	  ELSIF (#statStatus = #STATUS_COMMAND_ABORTED) AND (#statCommandAborted = FALSE) THEN // Commanded functionality has been aborted by another command
	    #statDone := FALSE;
	    #statBusy := FALSE;
	    #statActive := FALSE;
	    #statCommandAborted := TRUE;
	    #statError := FALSE;
	    #diagnostics.stateNumber := #statFBState;
	    #diagnostics.status := #statStatus;
	    #diagnostics.subFunctionStatus := #statSubfunctionStatus;
	    #diagnostics.additionalValue1 := #statAdditionalValue[1];
	    #diagnostics.additionalValue2 := #statAdditionalValue[2];
	    #statFBState := #FB_STATE_NO_PROCESSING; // Switch state machine to "no processing"
	    //Restore TO data
	    IF (#statReadyForNextCommand = FALSE) THEN
	      //only do if not done yet
	      "LKinCtrl_InitTODataRestore"(initTOData := #statInitTOData,
	                                   axesGroup := #axesGroup);
	    END_IF;
	    // Reset application specific outputs
	    #statReadyForNextCommand := FALSE;
	    #statCommandStep := #CMD_STEP_IDLE;
	    #statRemainingPathLength := -1.0;
	    
	  ELSIF (#tempExecute = FALSE) AND ((#statDone = TRUE) OR (#statError = TRUE) OR (#statCommandAborted = TRUE)) THEN // Reset outputs
	    #statDone := FALSE;
	    #statBusy := FALSE;
	    #statActive := FALSE;
	    #statCommandAborted := FALSE;
	    #statError := FALSE;
	    #statStatus := #STATUS_NO_CALL;
	    // Reset application specific outputs
	    #statReadyForNextCommand := FALSE;
	    #statCommandStep := #CMD_STEP_IDLE;
	    #statRemainingPathLength := -1.0;
	  END_IF;
	  
	  // Write static values to outputs
	  #done := #statDone;
	  #busy := #statBusy;
	  #active := #statActive;
	  #commandAborted := #statCommandAborted;
	  #error := #statError;
	  #status := #statStatus;
	  // Write application specific static values to outputs
	  #readyForNextCommand := #statReadyForNextCommand;
	  #commandStep := #statCommandStep;
	  #remainingPathLength := #statRemainingPathLength;
	END_REGION OUTPUTS
END_FUNCTION_BLOCK

FUNCTION "LKinCtrl_InitTODataStore" : "LKinCtrl_typePnPInitTOData"
TITLE = LKinCtrl_InitTODataStore
{ S7_Optimized_Access := 'TRUE' }
AUTHOR : 'handling.team.automation@siemens.com'
FAMILY : LKinCtrl
VERSION : 5.0
//Store specific TO data
   VAR_IN_OUT 
      axesGroup {InstructionName := 'TO_Kinematics'; LibVersion := '9.0'} : TO_Kinematics;   // Reference to axes group
   END_VAR


BEGIN
	//=============================================================================
	// SIEMENS AG
	// (c)Copyright 2023
	//-----------------------------------------------------------------------------
	// Library:       LKinCtrl
	// Tested with:   S7-1518TF-4 PN/DP, FW V3.1
	// Engineering:   TIA Portal V19
	// Restrictions:  ---
	// Requirements:  S7-1500T, FW V3.0
	// Functionality: Store specific TO data
	// Support: tech.team.motioncontrol@siemens.com
	// Note: Parameter comments are only available in language 'English (United States)'
	//-----------------------------------------------------------------------------
	// Change log table:
	// Version  Date       Expert in charge Changes applied
	// 01.00.00 21.09.2023 SF               First released version
	//=============================================================================
	
	//Blending length factor
	#LKinCtrl_InitTODataStore.factorBlendingLength := #axesGroup.Transition.FactorBlendingLength;
	//Orientation dynamics
	#LKinCtrl_InitTODataStore.orientationDefaults.velocity := #axesGroup.DynamicDefaults.Orientation.Velocity;
	#LKinCtrl_InitTODataStore.orientationDefaults.acceleration := #axesGroup.DynamicDefaults.Orientation.Acceleration;
	#LKinCtrl_InitTODataStore.orientationDefaults.deceleration := #axesGroup.DynamicDefaults.Orientation.Deceleration;
	#LKinCtrl_InitTODataStore.orientationDefaults.jerk := #axesGroup.DynamicDefaults.Orientation.Jerk;
END_FUNCTION

FUNCTION "LKinCtrl_CallMC_TrackConv" : Void
TITLE = LKinCtrl_CallMC_TrackConv
{ S7_Optimized_Access := 'TRUE' }
AUTHOR : 'handling.team.automation@siemens.com'
FAMILY : LKinCtrl
VERSION : 5.0
//Call given MC_TrackConveyorBelt instance
   VAR_INPUT 
      axis : DB_ANY;   // Axis input
      axesGroup {InstructionName := 'TO_Kinematics'; LibVersion := '9.0'} : TO_Kinematics;   // Kinematics input
   END_VAR

   VAR_IN_OUT 
      instTrackConveyorBelt {InstructionName := 'MC_TRACKCONVEYORBELT'; LibVersion := '9.0'} : MC_TRACKCONVEYORBELT;   // Instance of MC_TrackConveyorBelt to be called
   END_VAR

   VAR_TEMP 
      tempRefAxis {InstructionName := 'TO_PositioningAxis'; LibVersion := '9.0'} : REF_TO TO_PositioningAxis;   // Temporary reference to positioning axis
      tempRefEncoder {InstructionName := 'TO_ExternalEncoder'; LibVersion := '9.0'} : REF_TO TO_ExternalEncoder;   // Temporary reference to external encoder
      tempRefProxy {InstructionName := 'TO_LeadingAxisProxy'; LibVersion := '9.0'} : REF_TO TO_LeadingAxisProxy;   // Temporary reference to leading axis proxy
   END_VAR


BEGIN
	//================================================================================
	// SIEMENS AG
	// (c)Copyright 2023 All Rights Reserved
	//--------------------------------------------------------------------------------
	// Library: LKinCtrl
	// Tested with: S7-1517T-3 PN
	// Engineering: TIA Portal V18
	// Restrictions: -
	// Requirements: S7-1500T FW 3.0
	// Functionality: Call MC_TrackConveyorBelt
	// Support: tech.team.motioncontrol@siemens.com
	// Note: Parameter comments are only available in language 'English (United States)'
	//-----------------------------------------------------------------------------
	// Change log table:
	// Version    Date          Expert in charge    Changes applied
	// 01.00.00   11.01.2022    FR                  First released version
	//===========================================================================================
	
	CASE TypeOfDB(#axis) OF
	  TO_PositioningAxis, TO_SynchronousAxis:
	    #tempRefAxis ?= #axis;
	    IF #tempRefAxis = NULL THEN
	      // Error
	      RETURN;
	    END_IF;
	    
	    // call MC_TrackConveyorBelt
	    #instTrackConveyorBelt(AxesGroup := #axesGroup,
	                           ConveyorBelt := #tempRefAxis^);
	    
	  TO_ExternalEncoder:
	    #tempRefEncoder ?= #axis;
	    IF #tempRefEncoder = NULL THEN
	      // Error
	      RETURN;
	    END_IF;
	    
	    // call MC_TrackConveyorBelt
	    #instTrackConveyorBelt(AxesGroup := #axesGroup,
	                           ConveyorBelt := #tempRefEncoder^);
	    
	  TO_LeadingAxisProxy:
	    #tempRefProxy ?= #axis;
	    IF #tempRefProxy = NULL THEN
	      // Error
	      RETURN;
	    END_IF;
	    
	    // call MC_TrackConveyorBelt
	    #instTrackConveyorBelt(AxesGroup := #axesGroup,
	                           ConveyorBelt := #tempRefProxy^);
	    
	  ELSE
	    // invalid TO type
	    ;
	END_CASE;
	
	
END_FUNCTION

FUNCTION "LKinCtrl_CreateLinCmdSequence" : Word
TITLE = LKinCtrl_CreateLinCmdSequence
{ S7_Optimized_Access := 'TRUE' }
AUTHOR : 'handling.team.automation@siemens.com'
FAMILY : LKinCtrl
VERSION : 5.0
//Creation of the parameter for a linear command sequence
   VAR_INPUT 
      startParameter : "LKinCtrl_typePnPParameter";   // Depart vector parameter
      targetParameter : "LKinCtrl_typePnPParameter";   // Approach vector parameter
      position : Array[1..6] of LReal;   // Target position
      coordSystem : DInt;   // Target coordinate system, = 0: WCS, = 1: OCS[1], = 2: OCS[2], = 3: OCS[3]
      directionA : DInt;   // 1 - positive, 2 - negative, 3 - shortest way (Only necessary up to 4D Kinematics)
      bufferModeBegin : DInt;   // bufferMode for start of path motion
      transitionParameter : Array[1..5] of LReal;   // transitionParameter for start of path motion
      dynamics : "LKinCtrl_typePnPDynamics";   // Dynamics specification
      bufferModeTransition : DInt;   // bufferMode for blending post pick / pre target
      scaleMode : DInt;   // Scaling mode for start and target dynamics (0: disable, 1: velo, 2: velo and accel, 3: velo, accel and jerk)
   END_VAR

   VAR_OUTPUT 
      cmdPar : "LKinCtrl_typePnPLinCmdSeqParameter";   // Command parameters
      additionalValue : Array[1..5] of Word;   // Stati of subfunctions for diagnostics
   END_VAR

   VAR_IN_OUT 
      axesGroup {InstructionName := 'TO_Kinematics'; LibVersion := '9.0'} : TO_Kinematics;   // Reference to axes group
   END_VAR

   VAR_TEMP 
      tempUseStartDirection : Bool;
      tempUseTargetDirection : Bool;
      tempInt : Int;
      tempLreal : LReal;
      tempWord : Word;
      tempCase : Int;
      tempIntermStartPoint : Array[1..6] of LReal;
      tempIntermStartCoordSystem : DInt;
      tempIntermTargetPoint : Array[1..6] of LReal;
      tempIntermTargetCoordSystem : DInt;
      tempOrientationDimension : Int;
      tempStartPointFrame : "LKinCtrl_typeFrame";
      tempTargetPointFrame : "LKinCtrl_typeFrame";
      tempIntermPointFrame : "LKinCtrl_typeFrame";
      tempStartDirection : "LKinCtrl_typeCOff3DPoint";
      tempNormStartDirection : "LKinCtrl_typeCOff3DPoint";
      tempTargetDirection : "LKinCtrl_typeCOff3DPoint";
      tempNormTargetDirection : "LKinCtrl_typeCOff3DPoint";
      tempCmdPar : "LKinCtrl_typePnPLinCmdSeqParameter" := (((), [()], (), (), [-1.0], ((), (), ((), (), (), (), (), ()), ((), (), (), (), (), ())), (), ((), (), (), ()), (), ()), ((), [()], (), (), [-1.0], ((), (), ((), (), (), (), (), ()), ((), (), (), (), (), ())), (), ((), (), (), ()), (), ()), ((), [()], (), (), [-1.0], ((), (), ((), (), (), (), (), ()), ((), (), (), (), (), ())), (), ((), (), (), ()), (), ()), ((), [()], (), (), [-1.0], ((), (), ((), (), (), (), (), ()), ((), (), (), (), (), ())), (), ((), (), (), ()), (), ()), ((), [()], (), (), [-1.0], ((), (), ((), (), (), (), (), ()), ((), (), (), (), (), ())), (), ((), (), (), ()), (), ()), ());
      tempFactorBlendingLength : LReal;
      tempBlendingFromPreviousCmd : Bool;
      tempTransition1 : LReal;
      tempTransition2 : LReal;
      tempPossibleIntermTransition1 : LReal;
      tempPossibleIntermTransition2 : LReal;
      tempIntermTransition : LReal;
      tempAdditionalValue : Word;
      tempTimeOffset : LReal;
      tempEstimatedStartTransitionArea : LReal;
   END_VAR

   VAR CONSTANT 
      CASE_NO_VEC : Int := 1;   // Case: no start and target direction specified
      CASE_ONLY_TARGET_VEC : Int := 2;   // Case: only target direction specified
      CASE_ONLY_START_VEC : Int := 3;   // Case: only start direction specified
      CASE_ALL_VEC : Int := 4;   // Case: all directions specified
      INTERM_POINT_RATIO : LReal := 0.5;   // Intermediate point ratio
      STATUS_NO_ERR : Word := 16#0000;   // No error
      ERR_GET_TRACKING_INFO : Word := 16#9000;   // Error - Get tracking info
      ERR_BLENDING_NOT_ALLOWED : Word := 16#9001;   // Error - Blending is not allowed
      ERR_GET_ORI_DIMENSION : Word := 16#9002;   // Error - Get orientation dimension
      ERR_GET_LIN_POINT_DIST : Word := 16#9003;   // Error - Get linear point distance
      ERR_CALC_INTERM_POINT : Word := 16#9004;   // Error - Calculate intermediate point
      INTERM_POINT_MIN_BLENDING_FAC : LReal := 0.2;   // Minimum blending factor for intermediate point
      INTERM_POINT_MAX_BLENDING_FAC : LReal := 0.4;   // Maximum blending factor for intermediate point
   END_VAR


BEGIN
	//=============================================================================
	// SIEMENS AG
	// (c)Copyright 2023
	//-----------------------------------------------------------------------------
	// Library:       LKinCtrl
	// Tested with:   S7-1518TF-4 PN/DP, FW V3.1
	// Engineering:   TIA Portal V19
	// Restrictions:  ---
	// Requirements:  S7-1500T, FW V3.0
	// Functionality: This block is creating the parameter for a linear command sequence
	//                (Usage for LKinCtrl_MC_MovePickAndPlace...)
	// Support: tech.team.motioncontrol@siemens.com
	// Note: Parameter comments are only available in language 'English (United States)'
	//-----------------------------------------------------------------------------
	// Change log table:
	// Version  Date       Expert in charge Changes applied
	// 01.00.00 21.09.2023 SF               First released version
	//=============================================================================
	
	//Preset additional values
	FOR #tempInt := 1 TO 5 DO
	  #additionalValue[#tempInt] := #STATUS_NO_ERR;
	END_FOR;
	
	//Blending from previous command?
	#tempBlendingFromPreviousCmd := #bufferModeBegin <> "BM_BUFFERED";
	
	REGION GET_DIRECTION_INFO
	  //Save variable to vector data type
	  #tempStartDirection.x := #startParameter.direction[1];
	  #tempStartDirection.y := #startParameter.direction[2];
	  #tempStartDirection.z := #startParameter.direction[3];
	  //Get info about start vector
	  #tempUseStartDirection := NOT (#tempStartDirection.x = 0.0 AND #tempStartDirection.y = 0.0 AND #tempStartDirection.z = 0.0) AND #startParameter.workingHeight <> 0;
	  //Save variable to vector data type
	  #tempTargetDirection.x := #targetParameter.direction[1];
	  #tempTargetDirection.y := #targetParameter.direction[2];
	  #tempTargetDirection.z := #targetParameter.direction[3];
	  //Get info about target vector    
	  #tempUseTargetDirection := NOT (#tempTargetDirection.x = 0.0 AND #tempTargetDirection.y = 0.0 AND #tempTargetDirection.z = 0.0) AND #targetParameter.workingHeight <> 0;
	  
	  //Check if allowed
	  IF (#tempUseStartDirection = TRUE) AND (#tempBlendingFromPreviousCmd = TRUE) THEN
	    //not allowed
	    #LKinCtrl_CreateLinCmdSequence := #ERR_BLENDING_NOT_ALLOWED;
	    RETURN;
	  END_IF;
	  
	  //use target point in every case
	  #tempCmdPar.target.usePoint := TRUE;
	  
	  //Get info which points are used
	  IF (#tempUseStartDirection = FALSE) AND (#tempUseTargetDirection = FALSE) THEN
	    //No start and target direction specified
	    #tempCase := #CASE_NO_VEC;
	    //Set if points are used or not
	    #tempCmdPar.postStart.usePoint := FALSE;
	    #tempCmdPar.preTarget.usePoint := FALSE;
	    
	  ELSIF (#tempUseStartDirection = FALSE) THEN
	    //No start direction specified
	    #tempCase := #CASE_ONLY_TARGET_VEC;
	    //Set if points are used or not
	    #tempCmdPar.postStart.usePoint := FALSE;
	    #tempCmdPar.preTarget.usePoint := TRUE;
	    
	  ELSIF (#tempUseTargetDirection = FALSE) THEN
	    //No target direction specified
	    #tempCase := #CASE_ONLY_START_VEC;
	    //Set if points are used or not
	    #tempCmdPar.postStart.usePoint := TRUE;
	    #tempCmdPar.preTarget.usePoint := FALSE;
	    
	  ELSE
	    //All directions specified
	    #tempCase := #CASE_ALL_VEC;
	    //Set if points are used or not
	    #tempCmdPar.postStart.usePoint := TRUE;
	    #tempCmdPar.preTarget.usePoint := TRUE;
	    
	  END_IF;
	END_REGION REGION GET_DIRECTION_INFO
	
	REGION GET_START_INFO
	  //Get all start parameter depending on blending from previous cmd
	  //--> if blending would be active, kinematics would be still in motion
	  //--> start position and therefore the post start position cannot be determinded
	  IF (#tempBlendingFromPreviousCmd = FALSE) THEN
	    //Start point
	    //set parameter
	    #tempCmdPar.start.usePoint := TRUE; //Inidicates that parameter are valid
	    #tempCmdPar.start.directionA := #directionA;
	    #tempCmdPar.start.pathDynamics := #dynamics.path;
	    #tempCmdPar.start.dynamicAdaption := #dynamics.dynamicAdaption;
	    //get Start CS and tracking info 
	    #tempCmdPar.start.coordSystem := #axesGroup.StatusPath.CoordSystem;
	    #tempWord := "LKinCtrl_GetTrackingInfo"(coordSystem := #tempCmdPar.start.coordSystem,
	                                            axesGroup := #axesGroup,
	                                            trackingPar => #tempCmdPar.start.tracking);
	    IF (#tempWord.%X15 = TRUE) THEN
	      #LKinCtrl_CreateLinCmdSequence := #ERR_GET_TRACKING_INFO;
	      #additionalValue[1] := #tempWord;
	      RETURN;
	    END_IF;
	    //Start position
	    IF (#tempCmdPar.start.coordSystem = "CS_WCS") THEN
	      #tempCmdPar.start.position[1] := #axesGroup.TcpInWcs.x.Position;
	      #tempCmdPar.start.position[2] := #axesGroup.TcpInWcs.y.Position;
	      #tempCmdPar.start.position[3] := #axesGroup.TcpInWcs.z.Position;
	      #tempCmdPar.start.position[4] := #axesGroup.TcpInWcs.a.Position;
	      #tempCmdPar.start.position[5] := #axesGroup.TcpInWcs.b.Position;
	      #tempCmdPar.start.position[6] := #axesGroup.TcpInWcs.c.Position;
	    ELSIF (#tempCmdPar.start.coordSystem >= "CS_OCS1") AND (#tempCmdPar.start.coordSystem <= "CS_OCS3") THEN
	      #tempCmdPar.start.position[1] := #axesGroup.TcpInOcs[#tempCmdPar.start.coordSystem].x.Position;
	      #tempCmdPar.start.position[2] := #axesGroup.TcpInOcs[#tempCmdPar.start.coordSystem].y.Position;
	      #tempCmdPar.start.position[3] := #axesGroup.TcpInOcs[#tempCmdPar.start.coordSystem].z.Position;
	      #tempCmdPar.start.position[4] := #axesGroup.TcpInOcs[#tempCmdPar.start.coordSystem].a.Position;
	      #tempCmdPar.start.position[5] := #axesGroup.TcpInOcs[#tempCmdPar.start.coordSystem].b.Position;
	      #tempCmdPar.start.position[6] := #axesGroup.TcpInOcs[#tempCmdPar.start.coordSystem].c.Position;
	    END_IF;
	    
	    //PostStart point
	    IF (#tempCmdPar.postStart.usePoint = TRUE) THEN
	      //set parameter
	      #tempCmdPar.postStart.coordSystem := #tempCmdPar.start.coordSystem;
	      #tempCmdPar.postStart.directionA := #directionA;
	      #tempCmdPar.postStart.pathDynamics := "LKinCtrl_ScaleDynamics"(dynamicsIn := #dynamics.path,
	                                                                     scaleFactor := #startParameter.dynamicsFactor,
	                                                                     mode := #scaleMode);
	      #tempCmdPar.postStart.dynamicAdaption := #dynamics.dynamicAdaption;
	      #tempWord := "LKinCtrl_GetTrackingInfo"(coordSystem := #tempCmdPar.postStart.coordSystem,
	                                              axesGroup := #axesGroup,
	                                              trackingPar => #tempCmdPar.postStart.tracking);
	      IF (#tempWord.%X15 = TRUE) THEN
	        #LKinCtrl_CreateLinCmdSequence := #ERR_GET_TRACKING_INFO;
	        #additionalValue[1] := #tempWord;
	        RETURN;
	      END_IF;
	      //Norm start vector
	      IF (#tempUseStartDirection = TRUE) THEN
	        #tempNormStartDirection := "LKinCtrl_VecUnit"(#tempStartDirection);
	      ELSE
	        #tempNormStartDirection.x := 0.0;
	        #tempNormStartDirection.y := 0.0;
	        #tempNormStartDirection.z := 0.0;
	      END_IF;
	      //Calc point position
	      #tempCmdPar.postStart.position[1] := #tempCmdPar.start.position[1] + #tempNormStartDirection.x * (#startParameter.workingHeight); // + #start.transitionArea
	      #tempCmdPar.postStart.position[2] := #tempCmdPar.start.position[2] + #tempNormStartDirection.y * (#startParameter.workingHeight);
	      #tempCmdPar.postStart.position[3] := #tempCmdPar.start.position[3] + #tempNormStartDirection.z * (#startParameter.workingHeight);
	      #tempCmdPar.postStart.position[4] := #tempCmdPar.start.position[4];
	      #tempCmdPar.postStart.position[5] := #tempCmdPar.start.position[5];
	      #tempCmdPar.postStart.position[6] := #tempCmdPar.start.position[6];
	    END_IF;
	  ELSE
	    //Start parameter not valid
	    #tempCmdPar.start.usePoint := FALSE;
	  END_IF;
	END_REGION GET_START_INFO
	
	REGION GET_PRETARGET_INFO
	  //PreTarget point 
	  IF (#tempCmdPar.preTarget.usePoint = TRUE) THEN
	    //set parameter
	    //set buffer mode and transitionParameter below...
	    #tempCmdPar.preTarget.coordSystem := #coordSystem;
	    #tempCmdPar.preTarget.directionA := #directionA;
	    #tempCmdPar.preTarget.pathDynamics := #dynamics.path;
	    #tempCmdPar.preTarget.dynamicAdaption := #dynamics.dynamicAdaption;
	    #tempWord := "LKinCtrl_GetTrackingInfo"(coordSystem := #tempCmdPar.preTarget.coordSystem,
	                                            axesGroup := #axesGroup,
	                                            trackingPar => #tempCmdPar.preTarget.tracking);
	    IF (#tempWord.%X15 = TRUE) THEN
	      #LKinCtrl_CreateLinCmdSequence := #ERR_GET_TRACKING_INFO;
	      #additionalValue[1] := #tempWord;
	      RETURN;
	    END_IF;
	    //Norm start vector
	    IF (#tempUseTargetDirection = TRUE) THEN
	      #tempNormTargetDirection := "LKinCtrl_VecUnit"(#tempTargetDirection);
	    ELSE
	      #tempNormTargetDirection.x := 0.0;
	      #tempNormTargetDirection.y := 0.0;
	      #tempNormTargetDirection.z := 0.0;
	    END_IF;
	    //Calc point position
	    #tempCmdPar.preTarget.position[1] := #position[1] + #tempNormTargetDirection.x * (#targetParameter.workingHeight);
	    #tempCmdPar.preTarget.position[2] := #position[2] + #tempNormTargetDirection.y * (#targetParameter.workingHeight);
	    #tempCmdPar.preTarget.position[3] := #position[3] + #tempNormTargetDirection.z * (#targetParameter.workingHeight);
	    #tempCmdPar.preTarget.position[4] := #position[4];
	    #tempCmdPar.preTarget.position[5] := #position[5];
	    #tempCmdPar.preTarget.position[6] := #position[6];
	  END_IF;
	END_REGION GET_PRETARGET_INFO
	
	REGION GET_TARGET_INFO
	  //Target point
	  IF (#tempCmdPar.target.usePoint = TRUE) THEN
	    //set parameter
	    //set path dynamics, buffer mode and transitionParameter below...
	    #tempCmdPar.target.coordSystem := #coordSystem;
	    #tempCmdPar.target.directionA := #directionA;
	    #tempCmdPar.target.dynamicAdaption := #dynamics.dynamicAdaption;
	    #tempWord := "LKinCtrl_GetTrackingInfo"(coordSystem := #tempCmdPar.target.coordSystem,
	                                            axesGroup := #axesGroup,
	                                            trackingPar => #tempCmdPar.target.tracking);
	    IF (#tempWord.%X15 = TRUE) THEN
	      #LKinCtrl_CreateLinCmdSequence := #ERR_GET_TRACKING_INFO;
	      #additionalValue[1] := #tempWord;
	      RETURN;
	    END_IF;
	    #tempCmdPar.target.position := #position;
	  END_IF;
	END_REGION GET_TARGET_INFO
	
	REGION GET_INTERMEDIATE_INFO
	  //Check if intermediate point is necessary (motion between two tracked OCS)??
	  IF (#tempCmdPar.start.tracking.active = TRUE)
	    AND (#tempCmdPar.target.tracking.active = TRUE)
	    AND (#tempCmdPar.start.coordSystem <> #tempCmdPar.target.coordSystem)
	    AND (#tempCmdPar.start.coordSystem >= "CS_OCS1") AND (#tempCmdPar.start.coordSystem <= "CS_OCS3")
	    AND (#tempCmdPar.target.coordSystem >= "CS_OCS1") AND (#tempCmdPar.target.coordSystem <= "CS_OCS3")
	  THEN
	    IF (#tempBlendingFromPreviousCmd = TRUE) THEN
	      //not allowed
	      #LKinCtrl_CreateLinCmdSequence := #ERR_BLENDING_NOT_ALLOWED;
	      RETURN;
	    END_IF;
	    
	    //set parameter
	    //set buffer mode and transitionParameter below...
	    #tempCmdPar.intermediate.usePoint := TRUE;
	    #tempCmdPar.intermediate.coordSystem := "CS_WCS";
	    #tempCmdPar.intermediate.directionA := #tempCmdPar.target.directionA;
	    #tempCmdPar.intermediate.pathDynamics := #dynamics.path;
	    #tempCmdPar.intermediate.dynamicAdaption := #dynamics.dynamicAdaption;
	    
	    //set values for point calculation
	    IF (#tempCmdPar.postStart.usePoint = TRUE) THEN
	      #tempIntermStartPoint := #tempCmdPar.postStart.position;
	      #tempIntermStartCoordSystem := #tempCmdPar.postStart.coordSystem;
	    ELSE
	      #tempIntermStartPoint := #tempCmdPar.start.position;
	      #tempIntermStartCoordSystem := #tempCmdPar.start.coordSystem;
	    END_IF;
	    
	    IF (#tempCmdPar.preTarget.usePoint = TRUE) THEN
	      #tempIntermTargetPoint := #tempCmdPar.preTarget.position;
	      #tempIntermTargetCoordSystem := #tempCmdPar.preTarget.coordSystem;
	    ELSE
	      #tempIntermTargetPoint := #tempCmdPar.target.position;
	      #tempIntermTargetCoordSystem := #tempCmdPar.target.coordSystem;
	    END_IF;
	    
	    //get ori dimension according to kinematics
	    #tempWord := "LKinCtrl_GetOrientationDimension"(orientationDimension => #tempOrientationDimension,
	                                                    axesGroup := #axesGroup);
	    IF (#tempWord.%X15 = TRUE) THEN
	      #LKinCtrl_CreateLinCmdSequence := #ERR_GET_ORI_DIMENSION;
	      #additionalValue[1] := #tempWord;
	      RETURN;
	    END_IF;
	    
	    //Set additional time duration for reaching start point (= post start)
	    IF (#tempCmdPar.postStart.usePoint = TRUE) THEN
	      // Estimated transition area around post start
	      #tempEstimatedStartTransitionArea := LIMIT(MN := 0.0, IN := #startParameter.transitionArea, MX := #startParameter.workingHeight);
	      // Calc time for motion between start and post start
	      #tempWord := "LKinCtrl_PositioningTime"(distance := #startParameter.workingHeight, //Use complete length 
	                                              velocity := #tempCmdPar.postStart.pathDynamics.velocity * #axesGroup.Override.Velocity / 100.0,
	                                              acceleration := #tempCmdPar.postStart.pathDynamics.acceleration,
	                                              deceleration := #tempCmdPar.postStart.pathDynamics.deceleration,
	                                              jerk := #tempCmdPar.postStart.pathDynamics.jerk,
	                                              "time" => #tempTimeOffset);
	      //Fracture time - better estimation than calculate time with standstill at start of blending 
	      #tempTimeOffset := #tempTimeOffset * (1.0 - #tempEstimatedStartTransitionArea / #startParameter.workingHeight);
	      //Reset time if error occured
	      IF (#tempWord.%X15 = TRUE) THEN
	        #tempTimeOffset := 0.0;
	      END_IF;
	    ELSE
	      //No additional time
	      #tempTimeOffset := 0.0;
	      #tempEstimatedStartTransitionArea := 0.0;
	    END_IF;
	    
	    //calculate point
	    #tempWord := "LKinCtrl_CalcIntermediatePoint"(startPosition := #tempIntermStartPoint,
	                                                  targetPosition := #tempIntermTargetPoint,
	                                                  startCoordSystem := #tempIntermStartCoordSystem,
	                                                  targetCoordSystem := #tempIntermTargetCoordSystem,
	                                                  ratio := #INTERM_POINT_RATIO,
	                                                  orientationDimension := #tempOrientationDimension,
	                                                  directionA := #tempCmdPar.intermediate.directionA,
	                                                  pathDynamics := #tempCmdPar.intermediate.pathDynamics,
	                                                  timeOffset := #tempTimeOffset,
	                                                  intermediatePosition => #tempCmdPar.intermediate.position,
	                                                  additionalValue => #tempAdditionalValue,
	                                                  axesGroup := #axesGroup);
	    IF (#tempWord.%X15 = TRUE) THEN
	      #LKinCtrl_CreateLinCmdSequence := #ERR_CALC_INTERM_POINT;
	      #additionalValue[1] := #tempWord;
	      #additionalValue[2] := #tempAdditionalValue;
	      RETURN;
	    END_IF;
	  ELSE
	    #tempCmdPar.intermediate.usePoint := FALSE;
	  END_IF;
	END_REGION GET_INTERMEDIATE_INFO
	
	REGION CALC_LIN_POINT_DISTANCE
	  //Calc distance to previous point
	  #tempWord := "LKinCtrl_GetDistanceToPrevious"(cmdPar := #tempCmdPar,
	                                                axesGroup := #axesGroup);
	  IF (#tempWord.%X15 = TRUE) THEN
	    #LKinCtrl_CreateLinCmdSequence := #ERR_GET_LIN_POINT_DIST;
	    #additionalValue[1] := #tempWord;
	    RETURN;
	  END_IF;
	END_REGION CALC_LIN_POINT_DISTANCE
	
	REGION CALC_BLENDING_INFO
	  //get blending info and calc radii for all point
	  CASE #tempCase OF
	      
	    #CASE_NO_VEC:
	      
	      REGION BLENDING_NO_VEC
	        //Set path dynamics for target
	        #tempCmdPar.target.pathDynamics := #dynamics.path;
	        //Intermediate point necessary?
	        IF (#tempCmdPar.intermediate.usePoint = TRUE) THEN
	          //info: 3
	          //No blending from previous motion!
	          //Start to intermediate
	          #tempCmdPar.intermediate.bufferMode := "BM_BUFFERED";
	          //Blend to target with max radius (100%!)
	          #tempCmdPar.target.bufferMode := #bufferModeTransition;
	          #tempCmdPar.target.transitionParameter[1] := #tempCmdPar.target.distanceToPrevious * #INTERM_POINT_MAX_BLENDING_FAC;
	        ELSE
	          //info: 1 & 9
	          //Blend to target with start specification
	          #tempCmdPar.target.bufferMode := #bufferModeBegin;
	          #tempCmdPar.target.transitionParameter := #transitionParameter;
	        END_IF;
	      END_REGION BLENDING_NO_VEC
	      
	    #CASE_ONLY_TARGET_VEC:
	      
	      REGION BLENDING_ONLY_TARGET_VEC
	        //Set path dynamics for target
	        #tempCmdPar.target.pathDynamics := "LKinCtrl_ScaleDynamics"(dynamicsIn := #dynamics.path,
	                                                                    scaleFactor := #targetParameter.dynamicsFactor,
	                                                                    mode := #scaleMode);
	        
	        //Intermediate point necessary?
	        IF (#tempCmdPar.intermediate.usePoint = TRUE) THEN
	          //info: 4
	          //No blending from previous motion!
	          //Start to intermediate
	          #tempCmdPar.intermediate.bufferMode := "BM_BUFFERED";
	          //Blend to pretarget with max radius
	          //Get radius
	          #tempCmdPar.preTarget.bufferMode := #bufferModeTransition;
	          //is target transition overlaping minimum intermediate radius?
	          IF (#targetParameter.transitionArea > (1.0 - #INTERM_POINT_MIN_BLENDING_FAC) * #tempCmdPar.preTarget.distanceToPrevious) THEN
	            //yes - shorten transition area
	            #tempTransition1 := (1.0 - #INTERM_POINT_MIN_BLENDING_FAC) * #tempCmdPar.preTarget.distanceToPrevious;
	          ELSE
	            //no - use transition area from spec
	            #tempTransition1 := #targetParameter.transitionArea;
	          END_IF;
	          #tempCmdPar.preTarget.transitionParameter[1] := MIN(IN1 := #tempCmdPar.preTarget.distanceToPrevious - #tempTransition1, IN2 := #tempCmdPar.preTarget.distanceToPrevious * #INTERM_POINT_MAX_BLENDING_FAC);
	          //Blend to target with specified transition area
	          IF (#targetParameter.transitionArea <> 0.0) THEN
	            #tempCmdPar.target.bufferMode := #bufferModeTransition;
	            #tempCmdPar.target.transitionParameter[1] := #tempTransition1; //use from calculation above
	          ELSE
	            #tempCmdPar.target.bufferMode := "BM_BUFFERED";
	          END_IF;
	        ELSE
	          //info: 2 & 10
	          //Blend to pretarget with start specification
	          #tempCmdPar.preTarget.bufferMode := #bufferModeBegin;
	          #tempCmdPar.preTarget.transitionParameter[1] := #transitionParameter[1];
	          //Blend to target with specified transition area
	          IF (#targetParameter.transitionArea <> 0.0) THEN
	            #tempCmdPar.target.bufferMode := #bufferModeTransition;
	            #tempCmdPar.target.transitionParameter[1] := #targetParameter.transitionArea;
	          ELSE
	            #tempCmdPar.target.bufferMode := "BM_BUFFERED";
	          END_IF;
	        END_IF;
	      END_REGION BLENDING_ONLY_TARGET_VEC
	      
	    #CASE_ONLY_START_VEC:
	      //Always start from standstill, no blending from previous motion
	      
	      REGION BLENDING_ONLY_START_VEC
	        //Set path dynamics for target
	        #tempCmdPar.target.pathDynamics := #dynamics.path;
	        
	        //Intermediate point necessary?
	        IF (#tempCmdPar.intermediate.usePoint = TRUE) THEN
	          //info: 7
	          //no blending to post start
	          #tempCmdPar.postStart.bufferMode := "BM_BUFFERED";
	          //is start transition overlaping minimum intermediate radius?
	          IF (#startParameter.transitionArea > (1.0 - #INTERM_POINT_MIN_BLENDING_FAC) * #tempCmdPar.target.distanceToPrevious) THEN
	            //yes - shorten transition area
	            #tempTransition1 := (1.0 - #INTERM_POINT_MIN_BLENDING_FAC) * #tempCmdPar.target.distanceToPrevious;
	          ELSE
	            //no - use transition area from spec
	            #tempTransition1 := #startParameter.transitionArea;
	          END_IF;
	          IF (#startParameter.transitionArea <> 0.0) THEN
	            #tempCmdPar.intermediate.bufferMode := #bufferModeTransition;
	            #tempCmdPar.intermediate.transitionParameter[1] := #tempTransition1;
	          ELSE
	            #tempCmdPar.intermediate.bufferMode := "BM_BUFFERED";
	          END_IF;
	          //Blend to target with resulting radius
	          #tempCmdPar.target.bufferMode := #bufferModeTransition;
	          #tempCmdPar.target.transitionParameter[1] := MIN(IN1 := #tempCmdPar.target.distanceToPrevious - #tempTransition1, IN2 := #tempCmdPar.target.distanceToPrevious * #INTERM_POINT_MAX_BLENDING_FAC);
	        ELSE
	          //info: 5
	          //no blending to post start
	          #tempCmdPar.postStart.bufferMode := "BM_BUFFERED";
	          //Blend to target with start transition area
	          IF (#startParameter.transitionArea <> 0.0) THEN
	            #tempCmdPar.target.bufferMode := #bufferModeTransition;
	            #tempCmdPar.target.transitionParameter[1] := #startParameter.transitionArea;
	          ELSE
	            #tempCmdPar.target.bufferMode := "BM_BUFFERED";
	          END_IF;
	        END_IF;
	      END_REGION REGION BLENDING_ONLY_START_VEC
	      
	    #CASE_ALL_VEC:
	      //Always Start from standstill, no blending from previous motion
	      
	      REGION BLENDING_ALL_VEC
	        //Set path dynamics for target
	        #tempCmdPar.target.pathDynamics := "LKinCtrl_ScaleDynamics"(dynamicsIn := #dynamics.path,
	                                                                    scaleFactor := #targetParameter.dynamicsFactor,
	                                                                    mode := #scaleMode);
	        
	        //Intermediate point necessary?
	        IF (#tempCmdPar.intermediate.usePoint = TRUE) THEN
	          //info: 8
	          //no blending to post start
	          #tempCmdPar.postStart.bufferMode := "BM_BUFFERED";
	          
	          //is start transition overlaping minimum intermediate radius?
	          IF (#startParameter.transitionArea > (1.0 - #INTERM_POINT_MIN_BLENDING_FAC) * #tempCmdPar.intermediate.distanceToPrevious) THEN
	            //yes - shorten transition area
	            #tempTransition1 := (1.0 - #INTERM_POINT_MIN_BLENDING_FAC) * #tempCmdPar.intermediate.distanceToPrevious;
	          ELSE
	            //no - use transition area from spec
	            #tempTransition1 := #startParameter.transitionArea;
	          END_IF;
	          #tempPossibleIntermTransition1 := MIN(IN1 := #tempCmdPar.intermediate.distanceToPrevious - #tempTransition1, IN2 := #tempCmdPar.intermediate.distanceToPrevious * #INTERM_POINT_MAX_BLENDING_FAC);
	          
	          //is target transition overlaping minimum intermediate radius?
	          IF (#targetParameter.transitionArea > (1.0 - #INTERM_POINT_MIN_BLENDING_FAC) * #tempCmdPar.preTarget.distanceToPrevious) THEN
	            //yes - shorten transition area
	            #tempTransition2 := (1.0 - #INTERM_POINT_MIN_BLENDING_FAC) * #tempCmdPar.preTarget.distanceToPrevious;
	          ELSE
	            //no - use transition area from spec
	            #tempTransition2 := #targetParameter.transitionArea;
	          END_IF;
	          #tempPossibleIntermTransition2 := MIN(IN1 := #tempCmdPar.preTarget.distanceToPrevious - #tempTransition2, IN2 := #tempCmdPar.preTarget.distanceToPrevious * #INTERM_POINT_MAX_BLENDING_FAC);
	          
	          //Get minimum intermediate transition
	          #tempIntermTransition := MIN(IN1 := #tempPossibleIntermTransition1, IN2 := #tempPossibleIntermTransition2);
	          //adapt 1st if necessary
	          #tempTransition1 := MIN(IN1 := #tempTransition1, IN2 := #tempCmdPar.intermediate.distanceToPrevious - #tempIntermTransition);
	          //adapt 2nd if necessary
	          #tempTransition2 := MIN(IN1 := #tempTransition2, IN2 := #tempCmdPar.preTarget.distanceToPrevious - #tempIntermTransition);
	          
	          //Blend to intermediate with start transition area
	          IF (#startParameter.transitionArea <> 0.0) THEN
	            #tempCmdPar.intermediate.bufferMode := #bufferModeTransition;
	            #tempCmdPar.intermediate.transitionParameter[1] := #tempTransition1;
	          ELSE
	            #tempCmdPar.intermediate.bufferMode := "BM_BUFFERED";
	          END_IF;
	          
	          //Blend to pretarget with intermediate radius
	          #tempCmdPar.preTarget.bufferMode := #bufferModeTransition;
	          #tempCmdPar.preTarget.transitionParameter[1] := #tempIntermTransition;
	          //Blend to target with target transition area
	          IF (#targetParameter.transitionArea <> 0.0) THEN
	            #tempCmdPar.target.bufferMode := #bufferModeTransition;
	            #tempCmdPar.target.transitionParameter[1] := #tempTransition2;
	          ELSE
	            #tempCmdPar.target.bufferMode := "BM_BUFFERED";
	          END_IF;
	        ELSE
	          //info: 6
	          //no blending to post start
	          #tempCmdPar.postStart.bufferMode := "BM_BUFFERED";
	          //Check if blending radii are overlapping
	          IF ((#startParameter.transitionArea + #targetParameter.transitionArea) > #tempCmdPar.preTarget.distanceToPrevious)
	            AND ((#startParameter.transitionArea + #targetParameter.transitionArea) <> 0.0)
	          THEN
	            //Yes - shorten both radi by overplapping factor
	            #tempTransition1 := #startParameter.transitionArea * #tempCmdPar.preTarget.distanceToPrevious / (#startParameter.transitionArea + #targetParameter.transitionArea);
	            #tempTransition2 := #targetParameter.transitionArea * #tempCmdPar.preTarget.distanceToPrevious / (#startParameter.transitionArea + #targetParameter.transitionArea);
	          ELSE
	            //No - set areas directly
	            #tempTransition1 := #startParameter.transitionArea;
	            #tempTransition2 := #targetParameter.transitionArea;
	          END_IF;
	          //Blend to pretarget with start transition area
	          IF (#startParameter.transitionArea <> 0.0) THEN
	            #tempCmdPar.preTarget.bufferMode := #bufferModeTransition;
	            #tempCmdPar.preTarget.transitionParameter[1] := #tempTransition1;
	          ELSE
	            #tempCmdPar.preTarget.bufferMode := "BM_BUFFERED";
	          END_IF;
	          //Blend to target with target transition area
	          IF (#targetParameter.transitionArea <> 0.0) THEN
	            #tempCmdPar.target.bufferMode := #bufferModeTransition;
	            #tempCmdPar.target.transitionParameter[1] := #tempTransition2;
	          ELSE
	            #tempCmdPar.target.bufferMode := "BM_BUFFERED";
	          END_IF;
	        END_IF;
	      END_REGION BLENDING_ALL_VEC
	      
	    ELSE
	      ;
	  END_CASE;
	  
	END_REGION CALC_BLENDING_INFO
	
	REGION GET_NUMBER_OF_USED_CMD
	  //init value
	  #tempCmdPar.numberOfUsedCmd := 0;
	  IF (#tempCmdPar.postStart.usePoint = TRUE) THEN
	    #tempCmdPar.numberOfUsedCmd += 1;
	  END_IF;
	  IF (#tempCmdPar.intermediate.usePoint = TRUE) THEN
	    #tempCmdPar.numberOfUsedCmd += 1;
	  END_IF;
	  IF (#tempCmdPar.preTarget.usePoint = TRUE) THEN
	    #tempCmdPar.numberOfUsedCmd += 1;
	  END_IF;
	  IF (#tempCmdPar.target.usePoint = TRUE) THEN
	    #tempCmdPar.numberOfUsedCmd += 1;
	  END_IF;
	END_REGION GET_NUMBER_OF_USED_CMD
	
	REGION OUTPUT
	  //Everything done - copy to Out var
	  #cmdPar := #tempCmdPar;
	  #LKinCtrl_CreateLinCmdSequence := #STATUS_NO_ERR;
	END_REGION OUTPUT
	
	
END_FUNCTION

FUNCTION "LKinCtrl_GetTrackingInfo" : Word
TITLE = LKinCtrl_GetTrackingInfo
{ S7_Optimized_Access := 'TRUE' }
AUTHOR : 'handling.team.automation@siemens.com'
FAMILY : LKinCtrl
VERSION : 5.0
//Get information about active conveyor tracking on specific OCS
   VAR_INPUT 
      coordSystem : DInt;   // Coordiante system to be checked
   END_VAR

   VAR_OUTPUT 
      trackingPar : "LKinCtrl_typePnPTrackingProperties";   // Tracking info
   END_VAR

   VAR_IN_OUT 
      axesGroup {InstructionName := 'TO_Kinematics'; LibVersion := '9.0'} : TO_Kinematics;   // Reference to axes group
   END_VAR

   VAR_TEMP 
      tempInt : Int;
      tempLreal : LReal;
      tempWord : Word;
   END_VAR

   VAR CONSTANT 
      STATUS_NO_ERR : Word := 16#0000;   // No error
      ERR_GET_AXIS_MOTION_VEC : Word := 16#8000;   // Error - Get axis motion vector
   END_VAR


BEGIN
	//=============================================================================
	// SIEMENS AG
	// (c)Copyright 2023
	//-----------------------------------------------------------------------------
	// Library:       LKinCtrl
	// Tested with:   S7-1518TF-4 PN/DP, FW V3.1
	// Engineering:   TIA Portal V19
	// Restrictions:  ---
	// Requirements:  S7-1500T, FW V3.0
	// Functionality: This block returns information about active conveyor tracking of a OCS
	//                (Usage for LKinCtrl_MC_MovePickAndPlace...)
	// Support: tech.team.motioncontrol@siemens.com
	// Note: Parameter comments are only available in language 'English (United States)'
	//-----------------------------------------------------------------------------
	// Change log table:
	// Version  Date       Expert in charge Changes applied
	// 01.00.00 21.09.2023 SF               First released version
	//=============================================================================
	
	#LKinCtrl_GetTrackingInfo := #STATUS_NO_ERR;
	//preset active as false
	#trackingPar.active := FALSE;
	
	FOR #tempInt := "CS_OCS1" TO "CS_OCS3" DO
	  IF (#coordSystem = #tempInt) THEN
	    IF (#axesGroup.StatusConveyor[#tempInt].TrackingState > 0) THEN
	      //Tracking on start is actvie
	      #trackingPar.active := TRUE;
	      //Get CS frame (one by one due to system...)
	      #trackingPar.frame.x := #axesGroup.StatusOcsFrame[#tempInt].x;
	      #trackingPar.frame.y := #axesGroup.StatusOcsFrame[#tempInt].y;
	      #trackingPar.frame.z := #axesGroup.StatusOcsFrame[#tempInt].z;
	      #trackingPar.frame.a := #axesGroup.StatusOcsFrame[#tempInt].a;
	      #trackingPar.frame.b := #axesGroup.StatusOcsFrame[#tempInt].b;
	      #trackingPar.frame.c := #axesGroup.StatusOcsFrame[#tempInt].c;
	      //Get Obj position (one by one due to system...)
	      #trackingPar.objectPosition.x := #axesGroup.StatusConveyor[#tempInt].ObjectPosition.x;
	      #trackingPar.objectPosition.y := #axesGroup.StatusConveyor[#tempInt].ObjectPosition.y;
	      #trackingPar.objectPosition.z := #axesGroup.StatusConveyor[#tempInt].ObjectPosition.z;
	      #trackingPar.objectPosition.a := #axesGroup.StatusConveyor[#tempInt].ObjectPosition.a;
	      #trackingPar.objectPosition.b := #axesGroup.StatusConveyor[#tempInt].ObjectPosition.b;
	      #trackingPar.objectPosition.c := #axesGroup.StatusConveyor[#tempInt].ObjectPosition.c;
	      //Get conveyor axis motion values
	      #tempWord := "LKinCtrl_GetAxisMotionVec"(actualValues := FALSE,
	                                               position => #tempLreal,
	                                               velocity => #trackingPar.velocity,
	                                               acceleration => #tempLreal,
	                                               axis := #axesGroup.StatusConveyor[#tempInt].ConveyorBelt);
	      IF (#tempWord.%X15 = TRUE) THEN
	        #LKinCtrl_GetTrackingInfo := #ERR_GET_AXIS_MOTION_VEC;
	        RETURN; //TODO use EXIT for performance?
	      END_IF;
	      RETURN; //TODO use EXIT for performance?
	    ELSE
	      #trackingPar.active := FALSE;
	    END_IF;
	  END_IF;
	END_FOR;
END_FUNCTION

FUNCTION "LKinCtrl_GetAxisMotionVec" : Word
TITLE = LKinCtrl_GetAxisMotionVec
{ S7_Optimized_Access := 'TRUE' }
AUTHOR : 'handling.team.automation@siemens.com'
FAMILY : LKinCtrl
VERSION : 5.0
//Get axes motion vector (position, velocity, acceleration) of positioning axis / synchronous axis
   VAR_INPUT 
      actualValues : Bool;   // TRUE: Get actual axis values
      axis : DB_ANY;   // Reference to axis DB
   END_VAR

   VAR_OUTPUT 
      position : LReal;   // Axis position
      velocity : LReal;   // Axis velocity
      acceleration : LReal;   // Axis acceleration
   END_VAR

   VAR_TEMP 
      tempRefToPosAxis {InstructionName := 'TO_PositioningAxis'; LibVersion := '9.0'} : REF_TO TO_PositioningAxis;
   END_VAR

   VAR CONSTANT 
      STATUS_NO_ERR : Word := 16#0000;   // No error
      ERR_AXIS_TYPE : Word := 16#8000;   // Error - Invalid axis type (< PosAxis)
   END_VAR


BEGIN
	//=============================================================================
	// SIEMENS AG
	// (c)Copyright 2023
	//-----------------------------------------------------------------------------
	// Library:       LKinCtrl
	// Tested with:   S7-1518TF-4 PN/DP, FW V3.1
	// Engineering:   TIA Portal V19
	// Restrictions:  ---
	// Requirements:  S7-1500T, FW V3.0
	// Functionality: This block is returning the motion vector (position, velocity, acceleration)
	//                of an positioning axis / synchronous axis
	// Support: tech.team.motioncontrol@siemens.com
	// Note: Parameter comments are only available in language 'English (United States)'
	//-----------------------------------------------------------------------------
	// Change log table:
	// Version  Date       Expert in charge Changes applied
	// 01.00.00 21.09.2023 SF               First released version
	//=============================================================================
	
	//Preset output
	#LKinCtrl_GetAxisMotionVec := #STATUS_NO_ERR;
	
	//Axis type at least pos axis?
	#tempRefToPosAxis ?= #axis;
	
	IF (#tempRefToPosAxis <> NULL) THEN
	  //get actual or setpoint values?
	  IF (#actualValues = TRUE) THEN
	    #position := #tempRefToPosAxis^.ActualPosition;
	    #velocity := #tempRefToPosAxis^.ActualVelocity;
	    #acceleration := #tempRefToPosAxis^.ActualAcceleration;
	  ELSE
	    #position := #tempRefToPosAxis^.Position;
	    #velocity := #tempRefToPosAxis^.Velocity;
	    #acceleration := #tempRefToPosAxis^.Acceleration;
	  END_IF;
	ELSE
	  #LKinCtrl_GetAxisMotionVec := #ERR_AXIS_TYPE;
	END_IF;
	
	
END_FUNCTION

FUNCTION "LKinCtrl_ScaleDynamics" : "LKinCtrl_typePathDynamics"
TITLE = LKinCtrl_ScaleDynamics
{ S7_Optimized_Access := 'TRUE' }
AUTHOR : 'handling.team.automation@siemens.com'
FAMILY : LKinCtrl
VERSION : 5.0
//Scale dynamics values according to input factor
   VAR_INPUT 
      dynamicsIn : "LKinCtrl_typePathDynamics";   // Input dynamics
      scaleFactor : LReal;   // Scaling factor
      mode : DInt;   // Scaling mode for start and target dynamics (0: disable, 1: velo, 2: velo and accel, 3: velo, accel and jerk)
   END_VAR

   VAR CONSTANT 
      MODE_VELO_ACCEL : DInt := 2;   // Scale only velocity and acceleration
      MODE_VELO : DInt := 1;   // Scale only velocity
      MODE_DISALBE : DInt := 0;   // Scale nothing
   END_VAR


BEGIN
	//=============================================================================
	// SIEMENS AG
	// (c)Copyright 2023
	//-----------------------------------------------------------------------------
	// Library:       LKinCtrl
	// Tested with:   S7-1518TF-4 PN/DP, FW V3.1
	// Engineering:   TIA Portal V19
	// Restrictions:  ---
	// Requirements:  S7-1500T, FW V3.0
	// Functionality: Scale dynamics values (velocity, acceleration, deceleration and jerk)
	//                according to input factor
	// Support: tech.team.motioncontrol@siemens.com
	// Note: Parameter comments are only available in language 'English (United States)'
	//-----------------------------------------------------------------------------
	// Change log table:
	// Version  Date       Expert in charge Changes applied
	// 01.00.00 21.09.2023 SF               First released version
	//=============================================================================
	
	//Preset output
	#LKinCtrl_ScaleDynamics := #dynamicsIn;
	//Scale if necessary
	IF (#mode > #MODE_DISALBE) THEN
	  //Scale velocity
	  #LKinCtrl_ScaleDynamics.velocity := #dynamicsIn.velocity * #scaleFactor / 100.0;
	  IF (#mode > #MODE_VELO) THEN
	    //Scale acceleration 
	    #LKinCtrl_ScaleDynamics.acceleration := #dynamicsIn.acceleration * (#scaleFactor / 100.0) * (#scaleFactor / 100.0);
	    #LKinCtrl_ScaleDynamics.deceleration := #dynamicsIn.deceleration * (#scaleFactor / 100.0) * (#scaleFactor / 100.0);
	    IF (#mode > #MODE_VELO_ACCEL) THEN
	      //Scale jerk
	      #LKinCtrl_ScaleDynamics.jerk := #dynamicsIn.jerk * (#scaleFactor / 100.0) * (#scaleFactor / 100.0) * (#scaleFactor / 100.0);
	    END_IF;
	  END_IF;
	END_IF;
	
END_FUNCTION

FUNCTION "LKinCtrl_GetOrientationDimension" : Word
TITLE = LKinCtrl_GetOrientationDimension
{ S7_Optimized_Access := 'TRUE' }
AUTHOR : 'handling.team.automation@siemens.com'
FAMILY : LKinCtrl
VERSION : 5.0
//Get number of orientation axes for used kinematics object
   VAR_INPUT 
      axesGroup {InstructionName := 'TO_Kinematics'; LibVersion := '9.0'} : TO_Kinematics;   // Axes group
   END_VAR

   VAR_OUTPUT 
      orientationDimension : Int;   // 0: No orientation; 1: A; 2: A, B; 3: A, B, C
   END_VAR

   VAR CONSTANT 
      STATUS_NO_ERR : Word := 16#0000;   // No error
      ERR_KIN_TYPE_UNKNOWN : Word := 16#8000;   // Error - Kinematics type unkown
      ORI_NO_ORI : Int := 0;   // No orientation
      ORI_A : Int := 1;   // Orientation A
      ORI_AB : Int := 2;   // Orientation A, B
      ORI_ABC : Int := 3;   // Orientation A, B, C
   END_VAR


BEGIN
	//=============================================================================
	// SIEMENS AG
	// (c)Copyright 2023
	//-----------------------------------------------------------------------------
	// Library:       LKinCtrl
	// Tested with:   S7-1518TF-4 PN/DP, FW V3.1
	// Engineering:   TIA Portal V19
	// Restrictions:  ---
	// Requirements:  S7-1500T, FW V3.0
	// Functionality: This block is returning the Degrees of Freedom (DOF) for orientation
	//                of the input kinematics type
	// Support: tech.team.motioncontrol@siemens.com
	// Note: Parameter comments are only available in language 'English (United States)'
	//-----------------------------------------------------------------------------
	// Change log table:
	// Version  Date       Expert in charge Changes applied
	// 01.00.00 21.09.2023 SF               First released version
	//=============================================================================
	
	REGION KINEMATICS_TYPE
	  // Kinematics type
	  // 1 - Cartesian portal 2D
	  // 2 - Cartesian portal 2D with orientation
	  // 3 - Cartesian portal 3D
	  // 4 - Cartesian portal 3D with orientation
	  // 5 - Roller picker 2D
	  // 6 - Roller picker 2D with orientation
	  // 7 - Roller picker 3D (vertical)
	  // 8 - Roller picker 3D with orientation (vertical)
	  // 9 - Roller picker 3D with orientation (horizontal)
	  // 10 - SCARA 3D with orientation
	  // 11 - Articulated arm 2D
	  // 12 - Articulated arm 2D with orientation
	  // 13 - Articulated arm 3D
	  // 14 - Articulated arm 3D with orientation
	  // 15 - Delta picker 2D
	  // 16 - Delta picker 2D with orientation
	  // 17 - Delta picker 3D
	  // 18 - Delta picker 3D with orientation
	  // 19 - Reserved
	  // 20 - SCARA 2D with orientation
	  // 21 - Cylindrical robot 3D
	  // 22 - Cylindrical robot 3D with orientation
	  // 23 - Tripod 3D
	  // 24 - Tripod 3D with orientation
	  // 25 - 6-axis articulated arm with central hand (Kin+)
	  // 26 - Cartesian portal 3D with 2 orientations A, B (Kin+)
	  // 27 - Delta picker 3D with 2 orientations A, B (Kin+)
	  // 28 - Reserved
	  // 29 - Reserved
	  // 30 - Reserved
	  // 31 - User-defined 2D
	  // 32 - User-defined 2D with orientation A
	  // 33 - User-defined 3D
	  // 34 - User-defined 3D with orientation A
	  // 35 - User-defined kinematics systems 3D with 2 orientations A, B (Kin+)
	  // 36 - User-defined kinematics systems 3D with 3 orientations (Kin+)
	END_REGION
	
	//Preset
	#LKinCtrl_GetOrientationDimension := #STATUS_NO_ERR;
	
	CASE #axesGroup.Kinematics.TypeOfKinematics OF
	  1, 5, 11, 15, 31:  // 2D kinematics
	    #orientationDimension := #ORI_NO_ORI;
	  2, 6, 12, 16, 20, 32:  // 2D + orientation axis A;
	    #orientationDimension := #ORI_A;
	  3, 7, 13, 17, 21, 23, 33:  // 3D kinematics
	    #orientationDimension := #ORI_NO_ORI;
	  4, 8, 9, 10, 14, 18, 22, 24, 34:  // 3D + orientation axis A
	    #orientationDimension := #ORI_A;
	  26, 27, 35: // 3D + orientation axis A, B
	    #orientationDimension := #ORI_AB;
	  25, 36: // 3D + orientation axis A, B, C
	    #orientationDimension := #ORI_ABC;
	  ELSE  // invalid kinematics type
	    #LKinCtrl_GetOrientationDimension := #ERR_KIN_TYPE_UNKNOWN;
	END_CASE;
	
END_FUNCTION

FUNCTION "LKinCtrl_PositioningTime" : Word
TITLE = LKinCtrl_PositioningTime
{ S7_Optimized_Access := 'TRUE' }
AUTHOR : 'handling.team.automation@siemens.com'
FAMILY : LKinCtrl
VERSION : 5.0
//Calculate positioning time of motion profile
   VAR_INPUT 
      distance : LReal;   // Distance between start and end of motion command
      velocity : LReal;   // Velocity of motion command
      acceleration : LReal;   // Acceleration of motion command
      deceleration : LReal;   // Deceleration of motion command
      jerk : LReal;   // Jerk of motion command (Value = 0.0: Trapezoid velocity profile)
   END_VAR

   VAR_OUTPUT 
      "time" : LReal;   // Calculated time between start and end of motion command
   END_VAR

   VAR_TEMP 
      tempT02 : LReal;
      tempT1 : LReal;
      tempT2 : LReal;
      tempT3 : LReal;
      tempT4 : LReal;
      tempT46 : LReal;
      tempT5 : LReal;
      tempT6 : LReal;
      tempTGes : LReal;
      tempVelMax : LReal;
      tempDecMax : LReal;
      tempSetAcc : LReal;
      tempSetDec : LReal;
      tempAccDecMax : LReal;
      tempAccReach : LReal;
      tempAcc : LReal;
      tempDec : LReal;
      tempProfile : Int;
   END_VAR

   VAR CONSTANT 
      ERR_ACCEL_INVALID : Word := 16#8201;   // Acceleration value range exceeded (0.0 to 1.0e12)
      ERR_DECEL_INVALID : Word := 16#8202;   // Deceleration value range exceeded (0.0 to 1.0e12)
      ERR_DISTANCE_INVALID : Word := 16#8203;   // Distance value range exceeded (must be greater than 0.0)
      ERR_JERK_INVALID : Word := 16#8204;   // Jerk value range exceeded (0.0 to 1.0e12)
      ERR_VELOCITY_INVALID : Word := 16#8207;   // Velocity value range exceeded
   END_VAR


BEGIN
	//================================================================================
	// SIEMENS AG
	// (c)Copyright 2023 All Rights Reserved
	// -------------------------------------------------------------------------------
	// Library: LKinCtrl
	// Tested with: S7-1515T-2 PN
	// Engineering: TIA Portal V14
	// Restrictions: -
	// Requirements: S7-1500/S7-1500T FW 2.0
	// Functionality: Calculate time needed for MC_MoveAbsolute or MC_MoveRelative
	//                command
	// Support: tech.team.motioncontrol@siemens.com
	// Note: Parameter comments are only available in language 'English (United States)'
	// -------------------------------------------------------------------------------
	// Change log table:
	// Version   Date        Expert in charge  Changes applied
	// 01.00.00  16.08.2017  CR                First released version
	// 01.00.01  07.02.2020  KT                Error constants are now local (library conformance)
	// 01.00.02  02.03.2023  YT                Bug-fix: limit acceleration to not exceed
	//                                         the velocity input
	//================================================================================
	
	#LKinCtrl_PositioningTime := 16#0000;
	
	IF (#jerk < 0.0 OR #jerk > 1.0E12) THEN
	  #LKinCtrl_PositioningTime := #ERR_JERK_INVALID;
	  RETURN;
	ELSIF (#acceleration <= 0.0) OR (#acceleration > 1.0e12) THEN
	  #LKinCtrl_PositioningTime := #ERR_ACCEL_INVALID;
	  RETURN;
	ELSIF (#deceleration <= 0.0) OR (#deceleration > 1.0e12) THEN
	  #LKinCtrl_PositioningTime := #ERR_DECEL_INVALID;
	  RETURN;
	ELSIF (#distance <= 0.0) THEN
	  #LKinCtrl_PositioningTime := #ERR_DISTANCE_INVALID;
	  RETURN;
	ELSIF (#velocity <= 0.0) OR (#velocity > 1.0e12) THEN
	  #LKinCtrl_PositioningTime := #ERR_VELOCITY_INVALID;
	  RETURN;
	END_IF;
	
	IF (#jerk > 0.0) THEN
	  
	  #tempAccDecMax := (0.5 * #distance * (#jerk * #jerk)) ** (1.0 / 3.0);
	  
	  #tempVelMax := (0.25 * #jerk * (#distance * #distance)) ** (1.0 / 3.0);
	  
	  #tempAccReach := #velocity / SQRT_LREAL(MAX(IN1 := 0.0, IN2 := (#velocity / #jerk)));
	  
	  
	  #tempAcc := MIN(IN1 := #tempAccReach, IN2 := #acceleration, IN3 := #tempAccDecMax);
	  #tempDec := MIN(IN1 := #tempAccReach, IN2 := #deceleration, IN3 := #tempAccDecMax);
	  
	  IF (#tempAcc <= #tempDec) THEN
	    #tempSetAcc := #tempAcc;
	    #tempSetDec := #tempDec;
	  ELSE
	    #tempSetAcc := #tempDec;
	    #tempSetDec := #tempAcc;
	  END_IF;
	  
	  
	  IF #tempAccDecMax <= #acceleration OR #tempAccDecMax <= #deceleration OR #tempAccReach <= #acceleration OR #tempAccReach <= #deceleration THEN
	    IF (#tempAccDecMax <= #acceleration AND #tempAccDecMax <= #deceleration) OR (#tempAccReach <= #acceleration AND #tempAccReach <= #deceleration) THEN
	      IF #tempVelMax <= #velocity THEN
	        #tempProfile := 10;
	        #tempTGes := 4.0 * #tempAcc / #jerk;
	        
	      ELSE
	        #tempProfile := 20;
	        
	        #tempT4 := #distance / #velocity - (#tempAcc + #tempDec) * (#jerk * #velocity + #tempAcc * #tempDec) / (2.0 * #jerk * #tempAcc * #tempDec);
	        #tempTGes := 4.0 * #tempAcc / #jerk + #tempT4;
	      END_IF;
	      
	    ELSE
	      
	      #tempT46 := (SQRT_LREAL(MAX(IN1 := 0.0, IN2 := ((#tempSetAcc * #tempSetAcc) + 4.0 * #jerk * SQRT_LREAL(MAX(IN1 := 0.0, IN2 := (2.0 * #distance * #tempSetAcc)))))) - #tempSetAcc) / (2.0 * #jerk);
	      #tempDecMax := #jerk * #tempT46;
	      #tempT02 := #tempSetAcc / #jerk;
	      #tempVelMax := #tempDecMax * #tempT46;
	      
	      
	      IF (#tempVelMax <= #velocity) THEN
	        #tempProfile := 30;
	        
	        #tempT2 := (#jerk / #tempSetAcc) * ((#tempT46 * #tempT46) - (#tempT02 * #tempT02));
	        #tempTGes := 2.0 * #tempT02 + 2.0 * #tempT46 + #tempT2;
	        
	      ELSE
	        #tempProfile := 40;
	        #tempT1 := #tempT02;
	        #tempT2 := #velocity / #tempSetAcc - #tempT1;
	        #tempT5 := SQRT_LREAL(MAX(IN1 := 0.0, IN2 := (#velocity / #jerk)));
	        #tempT4 := #distance / #velocity - #tempT5 - (#velocity * #jerk + (#tempSetAcc * #tempSetAcc)) / (2.0 * #tempSetAcc * #jerk);
	        #tempTGes := 2.0 * #tempT1 + #tempT2 + #tempT4 + 2.0 * #tempT5;
	        
	      END_IF;
	    END_IF;
	  ELSE
	    
	    #tempT02 := #tempSetAcc / #jerk;
	    
	    #tempT46 := #tempSetDec / #jerk;
	    #tempT5 := SQRT_LREAL(MAX(IN1 := 0.0, IN2 := (((#tempSetAcc * #tempSetAcc) / (4.0 * (#jerk * #jerk))) + (2.0 * #distance * #tempSetAcc / (#tempSetDec * (#tempSetAcc + #tempSetDec)))))) - ((#tempSetAcc + 2.0 * #tempSetDec) / (2.0 * #jerk));
	    
	    #tempVelMax := #tempSetDec * (#tempT46 + #tempT5);
	    
	    IF (#tempVelMax <= #velocity) THEN
	      #tempProfile := 5;
	      #tempT1 := #tempSetAcc / #jerk;
	      #tempT2 := ((#tempSetDec * #tempSetDec) - (#tempSetAcc * #tempSetAcc) + #tempSetDec * #jerk * #tempT5) / (#tempSetAcc * #jerk);
	      #tempT5 := #tempSetDec / #jerk;
	      #tempT6 := SQRT_LREAL(MAX(IN1 := 0.0, IN2 := (((#tempSetAcc * #tempSetAcc) / (4.0 * (#jerk * #jerk))) + (2.0 * #distance * #tempSetAcc / (#tempSetDec * (#tempSetAcc + #tempSetDec)))))) - ((#tempSetAcc + 2.0 * #tempSetDec) / (2.0 * #jerk));
	      
	      #tempTGes := 2.0 * #tempT1 + #tempT2 + 2.0 * #tempT5 + #tempT6;
	      
	    ELSE
	      #tempProfile := 6;
	      #tempT1 := #tempSetAcc / #jerk;
	      #tempT5 := #tempSetDec / #jerk;
	      #tempT2 := #velocity / #tempSetAcc - #tempT02;
	      #tempT6 := #velocity / #tempSetDec - #tempT46;
	      #tempT4 := #distance / #velocity - (#tempSetAcc + #tempSetDec) * (#jerk * #velocity + #tempSetAcc * #tempSetDec) / (2.0 * #jerk * #tempSetAcc * #tempSetDec);
	      #tempTGes := 2.0 * #tempT1 + #tempT2 + #tempT4 + 2.0 * #tempT5 + #tempT6;
	    END_IF;
	  END_IF;
	ELSE
	  
	  #tempProfile := 100;
	  
	  #tempTGes := SQRT_LREAL(MAX(IN1 := 0.0, IN2 := ((#acceleration + #deceleration) * (2.0 * #distance) / (#acceleration * #deceleration))));
	  #tempVelMax := #tempTGes * (#acceleration * #deceleration) / (#acceleration + #deceleration);
	  
	  IF (#tempVelMax > #velocity) THEN
	    #tempProfile := 200;
	    #tempTGes := #distance / #velocity + (#velocity / 2.0) * (#acceleration + #deceleration) / (#acceleration * #deceleration);
	  END_IF;
	END_IF;
	
	#time := #tempTGes;
END_FUNCTION

FUNCTION "LKinCtrl_CalcIntermediatePoint" : Word
TITLE = LKinCtrl_CalcIntermediatePoint
{ S7_Optimized_Access := 'TRUE' }
AUTHOR : 'handling.team.automation@siemens.com'
FAMILY : LKinCtrl
VERSION : 5.0
//Calculation of the intermediate position (WCS) between a start and a target position (WCS or OCS)
   VAR_INPUT 
      startPosition : Array[1..6] of LReal;   // Start position in respective coordinate system
      targetPosition : Array[1..6] of LReal;   // Target position in respective coordinate system
      startCoordSystem : DInt;   // Start point coordiante system
      targetCoordSystem : DInt;   // Target point coordiante system
      ratio : LReal;   // Intermediate point ratio related to start point (0.05...0.95)
      orientationDimension : Int;   // 0 - no orientation, 1 - A, 2 - AB, 3 - ABC
      directionA : DInt;   // Only for orientationDimension = 1/A: 1 - positive, 2 - negative, 3 - shortest way
      pathDynamics : "LKinCtrl_typePathDynamics";   // Path dynamics for motion from start to target
      timeOffset : LReal;   // Estimated time for reaching start point in sec
   END_VAR

   VAR_OUTPUT 
      intermediatePosition : Array[1..6] of LReal;   // Intermediate position between start and target position
      additionalValue : Word;   // Additional value for diagnostics
   END_VAR

   VAR_IN_OUT 
      axesGroup {InstructionName := 'TO_Kinematics'; LibVersion := '9.0'} : TO_Kinematics;   // Reference to axes group
   END_VAR

   VAR_TEMP 
      tempLength : LReal;
      tempStartPointWCS : Array[1..6] of LReal;
      tempTargetPointWCS : Array[1..6] of LReal;
      tempIntermediateVec : "LKinCtrl_typeCOff3DPoint";
      tempIntermediateDir : "LKinCtrl_typeCOff3DPoint";
      tempIntermediatePointRatio : LReal;
      tempIntermediatePointWCS : Array[1..6] of LReal;
      tempWord : Word;
      tempTime : LReal;
      tempPosOffsetStart : LReal;
      tempPosOffsetTarget : LReal;
      tempDirVecStart : "LKinCtrl_typeCOff3DPoint";
      tempDirVecTarget : "LKinCtrl_typeCOff3DPoint";
      tempPreWeigthStart : LReal;
      tempPreWeigthTarget : LReal;
      tempVecScalarProd : LReal;
      tempVecAbs : LReal;
      tempVecAngle : LReal;
      tempStartPointFrame : "LKinCtrl_typeFrame";
      tempTargetPointFrame : "LKinCtrl_typeFrame";
      tempStartPointVelocity : LReal;
      tempTargetPointVelocity : LReal;
      tempStartCoordSystem : DInt;
      tempTargetCoordSystem : DInt;
      tempTrackingParStart : "LKinCtrl_typePnPTrackingProperties";
      tempTrackingParTarget : "LKinCtrl_typePnPTrackingProperties";
      tempStartCartesianPositionInitCS : Array[1..6] of LReal;
      tempTargetCartesianPositionInitCS : Array[1..6] of LReal;
      tempInt : Int;
      tempStartOri : "LKinCtrl_typePnPOrientationFrame";
      tempTargetOri : "LKinCtrl_typePnPOrientationFrame";
      tempIntermediateOri : "LKinCtrl_typePnPOrientationFrame";
      tempTimeOffset : LReal;
   END_VAR

   VAR CONSTANT 
      ORI_NO_ORI : Int := 0;   // No orientation
      ORI_A : Int := 1;   // Orientation A
      ORI_AB : Int := 2;   // Orientation A, B
      ORI_ABC : Int := 3;   // Orientation A, B, C
      CALC_TOL : LReal := 0.001;   // Calculation tolerance
      RATIO_MIN : LReal := 0.05;   // Minimum intermediate point ratio
      RATIO_MAX : LReal := 0.95;   // Maximum intermediate point ratio
      RADDEG : LReal := 57.2957795130823;   // Radians to degree
      PI : LReal := 3.14159265358979;   // Pi
      STATUS_NO_ERR : Word := 16#0000;   // No error
      ERR_EQUAL_POINTS : Word := 16#9000;   // Error - equal points
      ERR_INVALID_CS : Word := 16#9001;   // Error - invalid start or target coordSystem
      ERR_DYN_PROFILE : Word := 16#9002;   // Error - at profile calculation
      ERR_CREATE_ROT_VEC : Word := 16#9003;   // Error - at calculation of rotation vector
      ERR_CREATE_VEC_ANGLE : Word := 16#9004;   // Error - at calculation of rotation vector angle
      ERR_INVALID_ORI_DIM : Word := 16#9005;   // Error - orientation dimension invalid
      ERR_CALC_ORI : Word := 16#9006;   // Error - orientation calculation
      ERR_GET_TRACKING_INFO : Word := 16#9007;   // Error - at getting tracking information
      PRECONTROL_WEIGHT_FAC : LReal := 0.4;   // Tracking precontrol factor
   END_VAR


BEGIN
	//=============================================================================
	// SIEMENS AG
	// (c)Copyright 2023
	//-----------------------------------------------------------------------------
	// Library:       LKinCtrl
	// Tested with:   S7-1518TF-4 PN/DP, FW V3.1
	// Engineering:   TIA Portal V19
	// Restrictions:  ---
	// Requirements:  S7-1500T, FW V3.0
	// Functionality: This block is calculating the position of a intermediate position (WCS) 
	//                between a start and a target position (WCS or OCS) 
	// Support: tech.team.motioncontrol@siemens.com
	// Note: Parameter comments are only available in language 'English (United States)'
	//-----------------------------------------------------------------------------
	// Change log table:
	// Version  Date       Expert in charge Changes applied
	// 01.00.00 21.09.2023 SF               First released version
	//=============================================================================
	
	//Preset additional values
	#additionalValue := #STATUS_NO_ERR;
	
	REGION CHECK_INPUTS
	  //Check coord systems
	  IF (#startCoordSystem < "CS_WCS") OR (#startCoordSystem > "CS_OCS3")
	    OR (#targetCoordSystem < "CS_WCS") OR (#targetCoordSystem > "CS_OCS3")
	  THEN
	    #LKinCtrl_CalcIntermediatePoint := #ERR_INVALID_CS;
	    RETURN;
	  END_IF;
	  
	  // Limit intermediate point ratio betweenn MIN and MAX
	  #tempIntermediatePointRatio := LIMIT(MN := #RATIO_MIN, IN := #ratio, MX := #RATIO_MAX);
	  
	  // Check working heigth dim
	  IF (#orientationDimension < #ORI_NO_ORI) OR (#orientationDimension > #ORI_ABC) THEN
	    #LKinCtrl_CalcIntermediatePoint := #ERR_INVALID_ORI_DIM;
	    RETURN;
	  END_IF;
	  
	  // Time offset
	  IF (#timeOffset >= 0.0) THEN
	    #tempTimeOffset := #timeOffset;
	  END_IF;
	END_REGION
	
	REGION GET_FRAME_INFO
	  
	  //copy input position values (maybe add object position later, if in tracking...) from to internal format
	  #tempStartCartesianPositionInitCS := #startPosition;
	  #tempTargetCartesianPositionInitCS := #targetPosition;
	  
	  REGION START_FRAME
	    //Get info for start cs
	    #tempStartCoordSystem := #startCoordSystem;
	    IF (#tempStartCoordSystem <> "CS_WCS") THEN
	      //Get tracking info
	      #tempWord := "LKinCtrl_GetTrackingInfo"(coordSystem := #tempStartCoordSystem,
	                                              axesGroup := #axesGroup,
	                                              trackingPar => #tempTrackingParStart);
	      IF (#tempWord.%X15 = TRUE) THEN
	        #LKinCtrl_CalcIntermediatePoint := #ERR_GET_TRACKING_INFO;
	        #additionalValue := #tempWord;
	        RETURN;
	      END_IF;
	      //Tracking active?
	      IF (#tempTrackingParStart.active = TRUE) THEN
	        //Add object position
	        #tempStartCartesianPositionInitCS[1] += #tempTrackingParStart.objectPosition.x;
	        //CS velocity and frame
	        #tempStartPointVelocity := #tempTrackingParStart.velocity;
	        #tempStartPointFrame := #tempTrackingParStart.frame;
	      ELSE
	        //static OCS
	        #tempStartPointVelocity := 0.0;
	        #tempStartPointFrame.x := #axesGroup.StatusOcsFrame[#tempStartCoordSystem].x;
	        #tempStartPointFrame.y := #axesGroup.StatusOcsFrame[#tempStartCoordSystem].y;
	        #tempStartPointFrame.z := #axesGroup.StatusOcsFrame[#tempStartCoordSystem].z;
	        #tempStartPointFrame.a := #axesGroup.StatusOcsFrame[#tempStartCoordSystem].a;
	        #tempStartPointFrame.b := #axesGroup.StatusOcsFrame[#tempStartCoordSystem].b;
	        #tempStartPointFrame.c := #axesGroup.StatusOcsFrame[#tempStartCoordSystem].c;
	      END_IF;
	    ELSE
	      #tempStartPointVelocity := 0.0;
	      #tempStartPointFrame.x := 0.0;
	      #tempStartPointFrame.y := 0.0;
	      #tempStartPointFrame.z := 0.0;
	      #tempStartPointFrame.a := 0.0;
	      #tempStartPointFrame.b := 0.0;
	      #tempStartPointFrame.c := 0.0;
	    END_IF;
	  END_REGION START_FRAME
	  
	  REGION TARGET_FRAME
	    //Get info for target cs
	    #tempTargetCoordSystem := #targetCoordSystem;
	    IF (#tempTargetCoordSystem <> "CS_WCS") THEN
	      //Get tracking info
	      #tempWord := "LKinCtrl_GetTrackingInfo"(coordSystem := #tempTargetCoordSystem,
	                                              axesGroup := #axesGroup,
	                                              trackingPar => #tempTrackingParTarget);
	      IF (#tempWord.%X15 = TRUE) THEN
	        #LKinCtrl_CalcIntermediatePoint := #ERR_GET_TRACKING_INFO;
	        #additionalValue := #tempWord;
	        RETURN;
	      END_IF;
	      //Tracking active?
	      IF (#tempTrackingParTarget.active = TRUE) THEN
	        //Add object position
	        #tempTargetCartesianPositionInitCS[1] += #tempTrackingParTarget.objectPosition.x;
	        //CS velocity and frame
	        #tempTargetPointVelocity := #tempTrackingParTarget.velocity;
	        #tempTargetPointFrame := #tempTrackingParTarget.frame;
	      ELSE
	        //static OCS
	        #tempTargetPointVelocity := 0.0;
	        #tempTargetPointFrame.x := #axesGroup.StatusOcsFrame[#tempTargetCoordSystem].x;
	        #tempTargetPointFrame.y := #axesGroup.StatusOcsFrame[#tempTargetCoordSystem].y;
	        #tempTargetPointFrame.z := #axesGroup.StatusOcsFrame[#tempTargetCoordSystem].z;
	        #tempTargetPointFrame.a := #axesGroup.StatusOcsFrame[#tempTargetCoordSystem].a;
	        #tempTargetPointFrame.b := #axesGroup.StatusOcsFrame[#tempTargetCoordSystem].b;
	        #tempTargetPointFrame.c := #axesGroup.StatusOcsFrame[#tempTargetCoordSystem].c;
	      END_IF;
	    ELSE
	      #tempTargetPointVelocity := 0.0;
	      #tempTargetPointFrame.x := 0.0;
	      #tempTargetPointFrame.y := 0.0;
	      #tempTargetPointFrame.z := 0.0;
	      #tempTargetPointFrame.a := 0.0;
	      #tempTargetPointFrame.b := 0.0;
	      #tempTargetPointFrame.c := 0.0;
	    END_IF;
	  END_REGION TARGET_FRAME
	  
	END_REGION GET_TRACKING_INFO
	
	REGION FRAME_OCS_TO_WCS
	  // Frame first point -> WCS
	  IF (#tempStartCoordSystem <> "CS_WCS") THEN
	    "LKinCtrl_OcsToWcs"(ocsX := #tempStartPointFrame.x,
	                        ocsY := #tempStartPointFrame.y,
	                        ocsZ := #tempStartPointFrame.z,
	                        ocsA := #tempStartPointFrame.a,
	                        ocsB := #tempStartPointFrame.b,
	                        ocsC := #tempStartPointFrame.c,
	                        pointXOcs := #tempStartCartesianPositionInitCS[1],
	                        pointYOcs := #tempStartCartesianPositionInitCS[2],
	                        pointZOcs := #tempStartCartesianPositionInitCS[3],
	                        pointAOcs := #tempStartCartesianPositionInitCS[4],
	                        pointBOcs := #tempStartCartesianPositionInitCS[5],
	                        pointCOcs := #tempStartCartesianPositionInitCS[6],
	                        pointXWcs => #tempStartPointWCS[1],
	                        pointYWcs => #tempStartPointWCS[2],
	                        pointZWcs => #tempStartPointWCS[3],
	                        pointAWcs => #tempStartPointWCS[4],
	                        pointBWcs => #tempStartPointWCS[5],
	                        pointCWcs => #tempStartPointWCS[6]);
	  ELSE
	    #tempStartPointWCS := #tempStartCartesianPositionInitCS;
	  END_IF;
	  // Frame second point -> WCS
	  IF (#tempTargetCoordSystem <> "CS_WCS") THEN
	    "LKinCtrl_OcsToWcs"(ocsX := #tempTargetPointFrame.x,
	                        ocsY := #tempTargetPointFrame.y,
	                        ocsZ := #tempTargetPointFrame.z,
	                        ocsA := #tempTargetPointFrame.a,
	                        ocsB := #tempTargetPointFrame.b,
	                        ocsC := #tempTargetPointFrame.c,
	                        pointXOcs := #tempTargetCartesianPositionInitCS[1],
	                        pointYOcs := #tempTargetCartesianPositionInitCS[2],
	                        pointZOcs := #tempTargetCartesianPositionInitCS[3],
	                        pointAOcs := #tempTargetCartesianPositionInitCS[4],
	                        pointBOcs := #tempTargetCartesianPositionInitCS[5],
	                        pointCOcs := #tempTargetCartesianPositionInitCS[6],
	                        pointXWcs => #tempTargetPointWCS[1],
	                        pointYWcs => #tempTargetPointWCS[2],
	                        pointZWcs => #tempTargetPointWCS[3],
	                        pointAWcs => #tempTargetPointWCS[4],
	                        pointBWcs => #tempTargetPointWCS[5],
	                        pointCWcs => #tempTargetPointWCS[6]);
	  ELSE
	    #tempTargetPointWCS := #tempTargetCartesianPositionInitCS;
	  END_IF;
	END_REGION
	
	REGION MANIPULATE_POINTS
	  // Create direction vector
	  #tempIntermediateVec.x := #tempTargetPointWCS[1] - #tempStartPointWCS[1];
	  #tempIntermediateVec.y := #tempTargetPointWCS[2] - #tempStartPointWCS[2];
	  #tempIntermediateVec.z := #tempTargetPointWCS[3] - #tempStartPointWCS[3];
	  
	  // Estimate (linear) length between start and target point
	  #tempLength := "LKinCtrl_VecAbs"(#tempIntermediateVec);
	  IF (#tempLength <= 0.0) THEN
	    #LKinCtrl_CalcIntermediatePoint := #ERR_EQUAL_POINTS;
	    RETURN;
	  END_IF;
	  
	  //Calculate time based on linear distance and input dynamics
	  //not accounted, as not known:
	  //  - actual travelled distance
	  //  - velocity profile deviations due to dynamics adaption, orientation limitation etc...
	  #tempWord := "LKinCtrl_PositioningTime"(distance := #tempLength,
	                                          velocity := #pathDynamics.velocity * #axesGroup.Override.Velocity / 100.0,
	                                          acceleration := #pathDynamics.acceleration,
	                                          deceleration := #pathDynamics.deceleration,
	                                          jerk := #pathDynamics.jerk,
	                                          "time" => #tempTime);
	  IF (#tempWord.%X15 = TRUE) THEN
	    #LKinCtrl_CalcIntermediatePoint := #ERR_DYN_PROFILE;
	    #additionalValue := #tempWord;
	    RETURN;
	  END_IF;
	  
	  //Calculate position offsets for precontrolling intermediate point
	  #tempPosOffsetStart := (#tempTimeOffset) * #tempStartPointVelocity;
	  #tempPosOffsetTarget := (#tempTime + #tempTimeOffset) * #tempTargetPointVelocity;
	  
	  //Shift WCS points according to OCS speed, rotation and time
	  #tempWord := "LKinCtrl_VecFrameDir"(frame := #tempStartPointFrame,
	                                      directionVector => #tempDirVecStart);
	  IF (#tempWord.%X15 = TRUE) THEN
	    #LKinCtrl_CalcIntermediatePoint := #ERR_CREATE_ROT_VEC;
	    #additionalValue := #tempWord;
	    RETURN;
	  END_IF;
	  #tempWord := "LKinCtrl_VecFrameDir"(frame := #tempTargetPointFrame,
	                                      directionVector => #tempDirVecTarget);
	  IF (#tempWord.%X15 = TRUE) THEN
	    #LKinCtrl_CalcIntermediatePoint := #ERR_CREATE_ROT_VEC;
	    #additionalValue := #tempWord;
	    RETURN;
	  END_IF;
	  
	  //calc vector between frames
	  #tempVecScalarProd := "LKinCtrl_VecScalProd"(vIn1 := #tempDirVecStart,
	                                               vIn2 := #tempDirVecTarget);
	  #tempVecAbs := "LKinCtrl_VecAbs"(#tempDirVecStart) * "LKinCtrl_VecAbs"(#tempDirVecTarget);
	  IF (#tempVecAbs = 0.0) THEN
	    #LKinCtrl_CalcIntermediatePoint := #ERR_CREATE_VEC_ANGLE;
	    RETURN;
	  END_IF;
	  IF (ABS(#tempVecScalarProd / #tempVecAbs) > 1.0) THEN
	    #LKinCtrl_CalcIntermediatePoint := #ERR_CREATE_VEC_ANGLE;
	    RETURN;
	  END_IF;
	  #tempVecAngle := ACOS(#tempVecScalarProd / #tempVecAbs) * #RADDEG;
	  IF (#tempVecAngle > 180.0) THEN
	    #tempVecAngle := #tempVecAngle - 180.0;
	  END_IF;
	  //Set weigth of precontrol
	  #tempPreWeigthStart := 1.0;
	  #tempPreWeigthTarget := 1.0 - #PRECONTROL_WEIGHT_FAC * ABS(#tempVecAngle) / 180.0;
	  
	  //-> update tempTargetPointWCS and tempStartPointWCS and calc again
	  //point = point + normal direction vector * tempPosOffset...
	  #tempStartPointWCS[1] := #tempStartPointWCS[1] + #tempDirVecStart.x * #tempPosOffsetStart * #tempPreWeigthStart;
	  #tempStartPointWCS[2] := #tempStartPointWCS[2] + #tempDirVecStart.y * #tempPosOffsetStart * #tempPreWeigthStart;
	  #tempStartPointWCS[3] := #tempStartPointWCS[3] + #tempDirVecStart.z * #tempPosOffsetStart * #tempPreWeigthStart;
	  
	  #tempTargetPointWCS[1] := #tempTargetPointWCS[1] + #tempDirVecTarget.x * #tempPosOffsetTarget * #tempPreWeigthTarget;
	  #tempTargetPointWCS[2] := #tempTargetPointWCS[2] + #tempDirVecTarget.y * #tempPosOffsetTarget * #tempPreWeigthTarget;
	  #tempTargetPointWCS[3] := #tempTargetPointWCS[3] + #tempDirVecTarget.z * #tempPosOffsetTarget * #tempPreWeigthTarget;
	END_REGION
	
	REGION POINT_CALCULATION
	  REGION XYZ_COORD
	    // Create direction vector
	    #tempIntermediateVec.x := #tempTargetPointWCS[1] - #tempStartPointWCS[1];
	    #tempIntermediateVec.y := #tempTargetPointWCS[2] - #tempStartPointWCS[2];
	    #tempIntermediateVec.z := #tempTargetPointWCS[3] - #tempStartPointWCS[3];
	    
	    // Estimate (linear) length between start and target point
	    #tempLength := "LKinCtrl_VecAbs"(#tempIntermediateVec);
	    IF (#tempLength <= 0.0) THEN
	      #LKinCtrl_CalcIntermediatePoint := #ERR_EQUAL_POINTS;
	      RETURN;
	    END_IF;
	    
	    // Normalised direction vector
	    #tempIntermediateDir := "LKinCtrl_VecUnit"(#tempIntermediateVec);
	    #tempIntermediatePointWCS[1] := #tempStartPointWCS[1] + #tempLength * #tempIntermediatePointRatio * #tempIntermediateDir.x;
	    #tempIntermediatePointWCS[2] := #tempStartPointWCS[2] + #tempLength * #tempIntermediatePointRatio * #tempIntermediateDir.y;
	    #tempIntermediatePointWCS[3] := #tempStartPointWCS[3] + #tempLength * #tempIntermediatePointRatio * #tempIntermediateDir.z;
	  END_REGION
	  
	  REGION ABC_COORD   
	    //Get start orientation frame
	    #tempStartOri.a := #tempStartPointWCS[4];
	    #tempStartOri.b := #tempStartPointWCS[5];
	    #tempStartOri.c := #tempStartPointWCS[6];
	    //Get target orientation frame
	    #tempTargetOri.a := #tempTargetPointWCS[4];
	    #tempTargetOri.b := #tempTargetPointWCS[5];
	    #tempTargetOri.c := #tempTargetPointWCS[6];
	    //Calc intermediate orientation
	    IF (#orientationDimension = #ORI_A) THEN //orientation A
	      //Calc intermediate frame between start and target frame
	      #tempWord := "LKinCtrl_IntermediateOriA"(startOri := #tempStartOri,
	                                               targetOri := #tempTargetOri,
	                                               ratio := #tempIntermediatePointRatio,
	                                               directionA := #directionA,
	                                               intermediateOri := #tempIntermediateOri);
	    ELSIF (#orientationDimension = #ORI_AB) THEN //2 orientations AB
	      //Calc intermediate frame between start and target frame
	      #tempWord := "LKinCtrl_IntermediateOriAB"(startOri := #tempStartOri,
	                                                targetOri := #tempTargetOri,
	                                                ratio := #tempIntermediatePointRatio,
	                                                intermediateOri := #tempIntermediateOri);
	    ELSIF (#orientationDimension = #ORI_ABC) THEN //3 orientations ABC
	      //Calc intermediate frame between start and target frame
	      #tempWord := "LKinCtrl_IntermediateOriABC"(startOri := #tempStartOri,
	                                                 targetOri := #tempTargetOri,
	                                                 ratio := #tempIntermediatePointRatio,
	                                                 intermediateOri => #tempIntermediateOri);
	    ELSE //no orientation
	      #tempIntermediateOri.a := 0.0;
	      #tempIntermediateOri.b := 0.0;
	      #tempIntermediateOri.c := 0.0;
	    END_IF;
	    //Set intermediate point orientation in array format
	    #tempIntermediatePointWCS[4] := #tempIntermediateOri.a;
	    #tempIntermediatePointWCS[5] := #tempIntermediateOri.b;
	    #tempIntermediatePointWCS[6] := #tempIntermediateOri.c;
	    
	    //Check error
	    IF (#tempWord.%X15 = TRUE) THEN
	      #LKinCtrl_CalcIntermediatePoint := #ERR_CALC_ORI;
	      #additionalValue := #tempWord;
	      RETURN;
	    END_IF;
	  END_REGION
	END_REGION
	
	REGION RETURN
	  //Return point in array format
	  #intermediatePosition := #tempIntermediatePointWCS;
	  //Return 0 -> everything ok!
	  #LKinCtrl_CalcIntermediatePoint := #STATUS_NO_ERR;
	  
	END_REGION RETURN
END_FUNCTION

FUNCTION "LKinCtrl_VecFrameDir" : Word
TITLE = LKinCtrl_VecFrameDir
{ S7_Optimized_Access := 'TRUE' }
AUTHOR : 'handling.team.automation@siemens.com'
FAMILY : LKinCtrl
VERSION : 5.0
//Calculates a unit vector which represents the X-direction of a frame
   VAR_INPUT 
      frame : "LKinCtrl_typeFrame";   // Input frame
   END_VAR

   VAR_OUTPUT 
      directionVector : "LKinCtrl_typeCOff3DPoint";   // Direction vector
   END_VAR

   VAR_TEMP 
      tempRotMatrix : Array[1..3, 1..3] of LReal;
      tempRetError : Bool;
      tempRetStatus : Word;
      tempUnitVecIn : Array[1..3, 1..1] of LReal;
      tempUnitVecOut : Array[1..3, 1..1] of LReal;
   END_VAR


BEGIN
	//=============================================================================
	// SIEMENS AG
	// (c)Copyright 2023
	//-----------------------------------------------------------------------------
	// Library:       LKinCtrl
	// Tested with:   S7-1518TF-4 PN/DP, FW V3.1
	// Engineering:   TIA Portal V19
	// Restrictions:  ---
	// Requirements:  S7-1500T, FW V3.0
	// Functionality: Calculates a unit vector which represents the X-direction of a frame
	// Support: tech.team.motioncontrol@siemens.com
	// Note: Parameter comments are only available in language 'English (United States)'
	//-----------------------------------------------------------------------------
	// Change log table:
	// Version  Date       Expert in charge Changes applied
	// 01.00.00 21.09.2023 SF               First released version
	//=============================================================================
	
	#tempRetStatus := 16#0;
	
	//create rotation matrix
	"LKinCtrl_RotXYZ"(angleA := #frame.a,
	                  angleB := #frame.b,
	                  angleC := #frame.c,
	                  resultMatrix := #tempRotMatrix);
	
	//create unit vector (in x direction)
	#tempUnitVecIn[1, 1] := 1.0;
	#tempUnitVecIn[2, 1] := 0.0;
	#tempUnitVecIn[3, 1] := 0.0;
	
	//Rotate unit vector around rotation matrix
	"LKinCtrl_MatrixMultiplication"(error => #tempRetError,
	                                status => #tempRetStatus,
	                                matrix1 := #tempRotMatrix,
	                                matrix2 := #tempUnitVecIn,
	                                matrixResult := #tempUnitVecOut);
	
	//set outputs
	#directionVector.x := #tempUnitVecOut[1, 1];
	#directionVector.y := #tempUnitVecOut[2, 1];
	#directionVector.z := #tempUnitVecOut[3, 1];
	#LKinCtrl_VecFrameDir := #tempRetStatus;
END_FUNCTION

FUNCTION "LKinCtrl_IntermediateOriA" : Word
TITLE = LKinCtrl_IntermediateOriA
{ S7_Optimized_Access := 'TRUE' }
AUTHOR : 'handling.team.automation@siemens.com'
FAMILY : LKinCtrl
VERSION : 5.0
//Calculate intermediate orientation (A) between start and target orientation
   VAR_INPUT 
      startOri : "LKinCtrl_typePnPOrientationFrame";   // Start orientation frame
      targetOri : "LKinCtrl_typePnPOrientationFrame";   // Target orientation frame
      ratio : LReal;   // Intermediate point ratio
      directionA : DInt;   // 1 - positive, 2 - negative, 3 - shortest way
   END_VAR

   VAR_IN_OUT 
      intermediateOri : "LKinCtrl_typePnPOrientationFrame";   // Intermediate orientation frame
   END_VAR

   VAR_TEMP 
      tempTargetFrameA : LReal;
   END_VAR

   VAR CONSTANT 
      STATUS_NO_ERR : Word := 16#0000;   // No error
      ERR_DIRA_INVALID : Word := 16#9000;   // Error - Direction A invalid
   END_VAR


BEGIN
	//=============================================================================
	// SIEMENS AG
	// (c)Copyright 2023
	//-----------------------------------------------------------------------------
	// Library:       LKinCtrl
	// Tested with:   S7-1518TF-4 PN/DP, FW V3.1
	// Engineering:   TIA Portal V19
	// Restrictions:  ---
	// Requirements:  S7-1500T, FW V3.0
	// Functionality: Calc intermediate frame A between start and target A
	// Support: tech.team.motioncontrol@siemens.com
	// Note: Parameter comments are only available in language 'English (United States)'
	//-----------------------------------------------------------------------------
	// Change log table:
	// Version  Date       Expert in charge Changes applied
	// 01.00.00 21.09.2023 SF               First released version
	//=============================================================================
	
	//init value
	#tempTargetFrameA := #targetOri.a;
	
	//check direction A
	IF (#directionA = 1) THEN //positive direction
	  //add 360° to target position until it is bigger than start
	  WHILE (#tempTargetFrameA < #startOri.a) DO
	    #tempTargetFrameA += 360.0;
	  END_WHILE;
	ELSIF (#directionA = 2) THEN //negative direction
	  //sub 360° from target position until it is lower than start
	  WHILE (#tempTargetFrameA > #startOri.a) DO
	    #tempTargetFrameA -= 360.0;
	  END_WHILE;
	ELSIF (#directionA = 3) THEN //shortest distance
	  ; //do nothing - keep target A!
	ELSE
	  #LKinCtrl_IntermediateOriA := #ERR_DIRA_INVALID;
	  RETURN;
	END_IF;
	
	//calculate intermediate position
	#intermediateOri.a := "LKinCtrl_GetValueInRange"(#startOri.a + "LKinCtrl_GetValueInRange"(#tempTargetFrameA - #startOri.a) * #ratio);
	#intermediateOri.b := 0.0; //Set all other to zero
	#intermediateOri.c := 0.0; //Set all other to zero
	
	//set return value
	#LKinCtrl_IntermediateOriA := #STATUS_NO_ERR;
	
	
END_FUNCTION

FUNCTION "LKinCtrl_GetValueInRange" : LReal
TITLE = LKinCtrl_GetValueInRange
{ S7_Optimized_Access := 'TRUE' }
AUTHOR : 'handling.team.automation@siemens.com'
FAMILY : LKinCtrl
VERSION : 5.0
//Get value in range -180°...179.999° (Modulo 360°)
   VAR_INPUT 
      value : LReal;   // Value
   END_VAR

   VAR_TEMP 
      tempValue : LReal;
   END_VAR

   VAR CONSTANT 
      VAL_MIN : LReal := -180.0;   // Range minimum
      VAL_MAX : LReal := 179.999;   // Range maximum
      VAL_RANGE : LReal := 360.0;   // Range
      ERR_NO_ERR : Word := 16#0000;   // No error
   END_VAR


BEGIN
	//=============================================================================
	// SIEMENS AG
	// (c)Copyright 2023
	//-----------------------------------------------------------------------------
	// Library:       LKinCtrl
	// Tested with:   S7-1518TF-4 PN/DP, FW V3.1
	// Engineering:   TIA Portal V19
	// Restrictions:  ---
	// Requirements:  S7-1500T, FW V3.0
	// Functionality: Return input value in range -180°...179.999° (modulo 360°)
	// Support: tech.team.motioncontrol@siemens.com
	// Note: Parameter comments are only available in language 'English (United States)'
	//-----------------------------------------------------------------------------
	// Change log table:
	// Version  Date       Expert in charge Changes applied
	// 01.00.00 21.09.2023 SF               First released version
	//=============================================================================
	
	#tempValue := #value;
	IF (#tempValue > #VAL_MAX) THEN //above range?
	  WHILE (#tempValue > #VAL_MAX) DO
	    #tempValue := #tempValue - #VAL_RANGE;
	  END_WHILE;
	ELSIF (#tempValue < #VAL_MIN) THEN
	  WHILE (#tempValue < #VAL_MIN) DO //below range?
	    #tempValue := #tempValue + #VAL_RANGE;
	  END_WHILE;
	ELSE
	  ;//in range
	END_IF;
	#LKinCtrl_GetValueInRange := #tempValue;
END_FUNCTION

FUNCTION "LKinCtrl_IntermediateOriAB" : Word
TITLE = LKinCtrl_IntermediateOriAB
{ S7_Optimized_Access := 'TRUE' }
AUTHOR : 'handling.team.automation@siemens.com'
FAMILY : LKinCtrl
VERSION : 5.0
//Calculate intermediate orientation (A, B) between start and target orientation
   VAR_INPUT 
      startOri : "LKinCtrl_typePnPOrientationFrame";   // Start orientation frame
      targetOri : "LKinCtrl_typePnPOrientationFrame";   // Target orientation frame
      ratio : LReal;   // Intermediate point ratio
   END_VAR

   VAR_IN_OUT 
      intermediateOri : "LKinCtrl_typePnPOrientationFrame";   // Intermediate orientation frame
   END_VAR

   VAR_TEMP 
      temp1 : LReal;
      temp2 : LReal;
      tempDistB : Array[1..2] of LReal;
      tempDistRatio : Array[1..2] of LReal;
      tempDistA : LReal;
      tempPoleFrame1 : Array[1..2] of "LKinCtrl_typePnPOrientationFrame";
      tempPoleFrame2 : Array[1..2] of "LKinCtrl_typePnPOrientationFrame";
      tempDistSum : Array[1..2] of LReal;
      tempDistC : LReal;
      tempIndex : USInt;
      tempPole : LReal;
   END_VAR

   VAR CONSTANT 
      CALC_TOL : LReal := 0.001;   // Calculation tolerance
      STATUS_NO_ERR : Word := 16#0000;   // No error
      NORTHPOLE : USInt := 1;   // Move across northpole of orientation sphere
      SOUTHPOLE : USInt := 2;   // Move across southpole of orientation sphere
   END_VAR


BEGIN
	//=============================================================================
	// SIEMENS AG
	// (c)Copyright 2023
	//-----------------------------------------------------------------------------
	// Library:       LKinCtrl
	// Tested with:   S7-1518TF-4 PN/DP, FW V3.1
	// Engineering:   TIA Portal V19
	// Restrictions:  ---
	// Requirements:  S7-1500T, FW V3.0
	// Functionality: Calc intermediate frame A, B between start and target A, B
	// Support: tech.team.motioncontrol@siemens.com
	// Note: Parameter comments are only available in language 'English (United States)'
	//-----------------------------------------------------------------------------
	// Change log table:
	// Version  Date       Expert in charge Changes applied
	// 01.00.00 21.09.2023 SF               First released version
	//=============================================================================
	
	//regard C
	IF ABS(#targetOri.c - #startOri.c) < #CALC_TOL THEN //same C
	  #intermediateOri.a := "LKinCtrl_GetValueInRange"(#startOri.a + "LKinCtrl_GetValueInRange"(#targetOri.a - #startOri.a) * #ratio);
	  #intermediateOri.b := #startOri.b + (#targetOri.b - #startOri.b) * #ratio;
	  #intermediateOri.c := 0.0;
	ELSE //different C
	  //Distance for C (-180 or +180?)
	  #tempDistC := #targetOri.c - #startOri.c;
	  //Calculate frame at poles
	  FOR #tempIndex := #NORTHPOLE TO #SOUTHPOLE DO
	    //Specify pole motion
	    IF (#tempIndex = #NORTHPOLE) THEN
	      #tempPole := -90.0; //Check northpole motion
	    ELSE
	      #tempPole := 90.0; //Check southpole motion
	    END_IF;
	    
	    //Get distance ratio START -> POLE -> TARGET (Orientation B)
	    #temp1 := #tempPole - #startOri.b;
	    #temp2 := #tempPole - #targetOri.b;
	    #tempDistB[#tempIndex] := #temp1 + #temp2;
	    IF #tempDistB[#tempIndex] <> 0.0 THEN
	      #tempDistRatio[#tempIndex] := #temp1 / #tempDistB[#tempIndex];
	    ELSE
	      //Already at pole
	      #tempDistRatio[#tempIndex] := 0.0;
	    END_IF;
	    //Calculate estimated distance of A
	    #tempDistA := "LKinCtrl_GetValueInRange"(#targetOri.a - #startOri.a - #tempDistC);
	    // ---> Frames at Pole (A = ?; B = +90 or -90; C  = 0/-180)
	    #tempPoleFrame1[#tempIndex].a := "LKinCtrl_GetValueInRange"(#startOri.a + #tempDistA * #tempDistRatio[#tempIndex]);
	    #tempPoleFrame1[#tempIndex].b := #tempPole;
	    #tempPoleFrame1[#tempIndex].c := #startOri.c;
	    
	    #tempPoleFrame2[#tempIndex].a := "LKinCtrl_GetValueInRange"(#startOri.a + #tempDistA * #tempDistRatio[#tempIndex] - #tempDistC);
	    #tempPoleFrame2[#tempIndex].b := #tempPole;
	    #tempPoleFrame2[#tempIndex].c := #targetOri.c;
	    
	    //Calculate geometric distance for evalulation
	    #tempDistSum[#tempIndex] := SQRT((#tempPoleFrame1[#tempIndex].a - #startOri.a) ** 2 + (#tempPoleFrame1[#tempIndex].b - #startOri.b) ** 2)
	    + SQRT((#targetOri.a - #tempPoleFrame2[#tempIndex].a) ** 2 + (#targetOri.b - #tempPoleFrame2[#tempIndex].b) ** 2);
	  END_FOR;
	  
	  //Check for shortest distance
	  IF (#tempDistSum[#NORTHPOLE] < #tempDistSum[#SOUTHPOLE]) THEN
	    #tempIndex := #NORTHPOLE; //Move over northpole (-90°)
	  ELSE
	    #tempIndex := #SOUTHPOLE; //Move over southpole (+90°)
	  END_IF;
	  
	  //intermediate ratio <= distance ratio --> Calculation between START and POLE 1, else Calculation between POLE 2 and TARGET
	  IF (#ratio <= #tempDistRatio[#tempIndex]) AND (#tempDistRatio[#tempIndex] > 0.0) THEN
	    //Intermediate point is between start and pole
	    #intermediateOri.a := "LKinCtrl_GetValueInRange"(#startOri.a + "LKinCtrl_GetValueInRange"(#tempPoleFrame1[#tempIndex].a - #startOri.a) * #ratio / #tempDistRatio[#tempIndex]);
	    #intermediateOri.b := #startOri.b + (#tempPoleFrame1[#tempIndex].b - #startOri.b) * #ratio / #tempDistRatio[#tempIndex];
	    #intermediateOri.c := #startOri.c;
	  ELSE
	    //Intermediate point is between pole and target
	    #intermediateOri.a := "LKinCtrl_GetValueInRange"(#tempPoleFrame2[#tempIndex].a + "LKinCtrl_GetValueInRange"(#targetOri.a - #tempPoleFrame2[#tempIndex].a) * (1.0 - #tempDistRatio[#tempIndex] - #ratio) / (1.0 - #tempDistRatio[#tempIndex]));
	    #intermediateOri.b := #tempPoleFrame2[#tempIndex].b + (#targetOri.b - #tempPoleFrame2[#tempIndex].b) * (1.0 - #tempDistRatio[#tempIndex] - #ratio) / (1.0 - #tempDistRatio[#tempIndex]);
	    #intermediateOri.c := #tempPoleFrame2[#tempIndex].c;
	  END_IF;
	END_IF;
	//set return value
	#LKinCtrl_IntermediateOriAB := #STATUS_NO_ERR;
	
	
END_FUNCTION

FUNCTION "LKinCtrl_IntermediateOriABC" : Word
TITLE = LKinCtrl_IntermediateOriABC
{ S7_Optimized_Access := 'TRUE' }
AUTHOR : 'handling.team.automation@siemens.com'
FAMILY : LKinCtrl
VERSION : 5.0
//Calculate intermediate orientation (A, B, C) between start and target orientation
   VAR_INPUT 
      startOri : "LKinCtrl_typePnPOrientationFrame";   // Start orientation frame
      targetOri : "LKinCtrl_typePnPOrientationFrame";   // Target orientation frame
      ratio : LReal;   // Intermediate point ratio
   END_VAR

   VAR_OUTPUT 
      intermediateOri : "LKinCtrl_typePnPOrientationFrame";   // Intermediate orientation frame
   END_VAR

   VAR_TEMP 
      tempMat1R2 : Array[1..3, 1..3] of LReal;
      tempMat0R1T : Array[1..3, 1..3] of LReal;
      tempMat0R1 : Array[1..3, 1..3] of LReal;
      tempMat0R2 : Array[1..3, 1..3] of LReal;
      tempMat1R3 : Array[1..3, 1..3] of LReal;
      tempMat0R3 : Array[1..3, 1..3] of LReal;
      tempRotationAngleRad : LReal;
      tempRotationAngle : LReal;
      tempRotationVec : "LKinCtrl_typeCOff3DPoint";
      tempRotationVecUnit : "LKinCtrl_typeCOff3DPoint";
      temp1 : LReal;
      tempError : Bool;
      tempStatus : Word;
   END_VAR

   VAR CONSTANT 
      STATUS_NO_ERR : Word := 16#0000;   // No error
      ERR_MATRIX_MUL : Word := 16#9000;   // Error - at matrix multiplication
   END_VAR


BEGIN
	//=============================================================================
	// SIEMENS AG
	// (c)Copyright 2023
	//-----------------------------------------------------------------------------
	// Library:       LKinCtrl
	// Tested with:   S7-1518TF-4 PN/DP, FW V3.1
	// Engineering:   TIA Portal V19
	// Restrictions:  ---
	// Requirements:  S7-1500T, FW V3.0
	// Functionality: Calc intermediate frame A, B, C between start and target A, B, C
	// Support: tech.team.motioncontrol@siemens.com
	// Note: Parameter comments are only available in language 'English (United States)'
	//-----------------------------------------------------------------------------
	// Change log table:
	// Version  Date       Expert in charge Changes applied
	// 01.00.00 21.09.2023 SF               First released version
	//=============================================================================
	
	//Create Matrix 0R2
	"LKinCtrl_RotXYZ"(angleA := #targetOri.a,
	                  angleB := #targetOri.b,
	                  angleC := #targetOri.c,
	                  resultMatrix := #tempMat0R2);
	//Create Matrix 0R1_T
	"LKinCtrl_RotXYZTranspose"(angleA := #startOri.a,
	                           angleB := #startOri.b,
	                           angleC := #startOri.c,
	                           resultMatrix := #tempMat0R1T);
	//Create Matrix OR1
	"LKinCtrl_RotXYZ"(angleA := #startOri.a,
	                  angleB := #startOri.b,
	                  angleC := #startOri.c,
	                  resultMatrix := #tempMat0R1);
	//Create Matrix 1R2 = 0R1_T*0R2
	"LKinCtrl_MatrixMultiplication"(error => #tempError,
	                                status => #tempStatus,
	                                matrix1 := #tempMat0R1T,
	                                matrix2 := #tempMat0R2,
	                                matrixResult := #tempMat1R2);
	IF (#tempError = TRUE) THEN
	  #LKinCtrl_IntermediateOriABC := #ERR_MATRIX_MUL;
	  RETURN;
	END_IF;
	//Create r, Phi
	"LKinCtrl_RotMatrixToRotVec"(rotMatrix := #tempMat1R2,
	                             rotVector => #tempRotationVecUnit,
	                             rotAngle => #tempRotationAngle);
	//Create 1R3 from r, Phi*ratio
	"LKinCtrl_RotVecToRotMatrix"(rotVector := #tempRotationVecUnit,
	                             rotAngle := #tempRotationAngle * #ratio,
	                             rotMatrix => #tempMat1R3);
	//Create 0R3 = 0R1 * 1R3
	"LKinCtrl_MatrixMultiplication"(error => #tempError,
	                                status => #tempStatus,
	                                matrix1 := #tempMat0R1,
	                                matrix2 := #tempMat1R3,
	                                matrixResult := #tempMat0R3);
	IF (#tempError = TRUE) THEN
	  #LKinCtrl_IntermediateOriABC := #ERR_MATRIX_MUL;
	  RETURN;
	END_IF;
	//Get A, B, C from 0R3
	"LKinCtrl_InvRotXYZ"(A => #intermediateOri.a,
	                     B => #intermediateOri.b,
	                     C => #intermediateOri.c,
	                     rotMatrix := #tempMat0R3);
	//set return value
	#LKinCtrl_IntermediateOriABC := #STATUS_NO_ERR;
	
	
END_FUNCTION

FUNCTION "LKinCtrl_RotMatrixToRotVec" : Void
TITLE = LKinCtrl_RotMatrixToRotVec
{ S7_Optimized_Access := 'TRUE' }
AUTHOR : 'handling.team.automation@siemens.com'
FAMILY : LKinCtrl
VERSION : 5.0
//Calculate rotation vector and angle from rotation matrix
   VAR_INPUT 
      rotMatrix : Array[1..3, 1..3] of LReal;   // Rotation matrix
   END_VAR

   VAR_OUTPUT 
      rotVector : "LKinCtrl_typeCOff3DPoint";   // Rotation vector
      rotAngle : LReal;   // Rotation angle
   END_VAR

   VAR_TEMP 
      tempR1 : LReal;
      tempR2 : LReal;
      tempR3 : LReal;
      tempResult1 : LReal;
      tempRotAngle : LReal;
      tempRadDeg : LReal;
   END_VAR

   VAR CONSTANT 
      PI : LReal := 3.14159265358979;   // Pi
      CALC_TOL : LReal := 0.001;   // Tolerance
   END_VAR


